RoboDK station: wcs_plc_20240513_133800.rdk

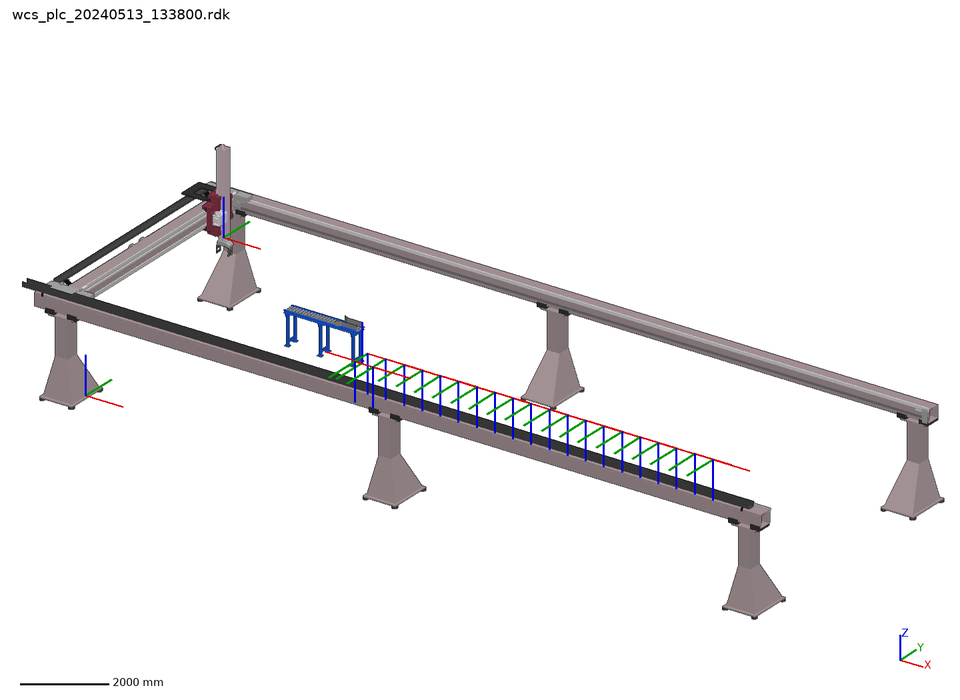
[picture v0: the station drawn from its stored meshes, robots at their saved joint values, targets as dots, program paths as lines]
Station wcs_plc_20240513_133800 (saved by RoboDK 5.6.8). Poses are relative to the parent item; angles as X-Y-Z fixed-axis rotations.
Station parameters (name, value as stored): TAGS, ['Milling']
  - frame conveyor Base IN at (4133.67, 4957.34, 0) mm, rotated rx 0 ry 0 rz 180 deg
    - robot conveyor IN: 1 axes
        modified DH rows (alpha deg, a mm, theta deg, d mm): 0, 0, 0, 0 linear
        base shift (0, 0, 0) mm, rotated rx 0 ry 90 rz 0 deg
        joint limits [-99999] to [9999999]; home [0]; saved at [1000]
      - tool conveyor_TCP_IN, TCP at (160, 110, 135) mm, rotated rx -180 ry 0 rz -180 deg
    - target con_pitch_IN (joint target) at (1000, 0, 880) mm; joints [1000, 0, 0] of conveyor IN
    - target con_home_IN (joint target) at (160, 110, 1015) mm, rotated rx -180 ry 0 rz -180 deg; joints [0] of conveyor IN
  - frame gantry Base at (0, 0, 0) mm
    - robot gantry: 3 axes
        modified DH rows (alpha deg, a mm, theta deg, d mm): 0, 0, 0, 0 linear; 90, 0, 90, 0 linear; 90, 0, 0, 0 linear
        base shift (0, 0, 0) mm, rotated rx 0 ry -90 rz 180 deg
        joint limits [-5, -5, -5] to [18000, 5000, 1500]; home [0, 0, 0]; saved at [0, 0, 0]
      - frame gripper Base at (0, 0, 0) mm, rotated rx -180 ry 0 rz 0 deg
        - robot gripper: 1 axes
            modified DH rows (alpha deg, a mm, theta deg, d mm): 0, 0, 0, 0 linear
            base shift (0, 0, 0) mm, rotated rx 0 ry 90 rz 0 deg
            joint limits [-200] to [0]; home [0]; saved at [-55]
        - target close_gripper (joint target) at (-121.33, 5507.34, 1743.56) mm; joints [-55] of gripper
        - target open_gripper (joint target) at (0, 0, 0) mm; joints [0, 0, 0] of gripper
      - tool gripper_TCP, TCP at (0, 0, 260) mm
    - target gantry_home (joint target) at (-66.33, 5507.34, 1483.56) mm, rotated rx 180 ry 0 rz 0 deg; joints [0, 0, 0] of gantry
    - target UP_pickup (joint target) at (3973.67, 4847.34, 1483.56) mm, rotated rx 180 ry 0 rz 0 deg; joints [4040, 660, 0] of gantry
    - target IN_pickup (joint target) at (3973.67, 4847.34, 1015) mm, rotated rx -180 ry 0 rz 0 deg; joints [4040, 660, 468.564] of gantry
    - target Target 6 (joint target) at (4133.67, 4957.34, 433.56) mm, rotated rx 180 ry 0 rz 0 deg; joints [4200, 550, 1050] of gantry
    - target Target 7 (Cartesian target) at (10933.67, 1007.34, 433.56) mm, rotated rx 180 ry 0 rz 0 deg; joints [11000, 4500, 1050] of gantry
    - folder pallet
      - frame TeachingPoints_01-01-01 at (4633.67, 4457.34, 568.56) mm, rotated rx 180 ry 0 rz 0 deg
        - target Point_01-01-01 (Cartesian target) at (0, 0, 0) mm; joints [4700, 1050, 915] of gantry
      - frame TeachingPoints_02-01-01 at (5133.67, 4457.34, 568.56) mm, rotated rx 180 ry 0 rz 0 deg
        - target Point_02-01-01 (Cartesian target) at (0, 0, 0) mm; joints [5200, 1050, 915] of gantry
      - frame TeachingPoints_03-01-01 at (5633.67, 4457.34, 568.56) mm, rotated rx 180 ry 0 rz 0 deg
        - target Point_03-01-01 (Cartesian target) at (0, 0, 0) mm; joints [5700, 1050, 915] of gantry
      - frame TeachingPoints_04-01-01 at (6133.67, 4457.34, 568.56) mm, rotated rx 180 ry 0 rz 0 deg
        - target Point_04-01-01 (Cartesian target) at (0, 0, 0) mm; joints [6200, 1050, 915] of gantry
      - frame TeachingPoints_05-01-01 at (6633.67, 4457.34, 568.56) mm, rotated rx 180 ry 0 rz 0 deg
        - target Point_05-01-01 (Cartesian target) at (0, 0, 0) mm; joints [6700, 1050, 915] of gantry
      - frame TeachingPoints_06-01-01 at (7133.67, 4457.34, 568.56) mm, rotated rx 180 ry 0 rz 0 deg
        - target Point_06-01-01 (Cartesian target) at (0, 0, 0) mm; joints [7200, 1050, 915] of gantry
      - frame TeachingPoints_07-01-01 at (7633.67, 4457.34, 568.56) mm, rotated rx 180 ry 0 rz 0 deg
        - target Point_07-01-01 (Cartesian target) at (0, 0, 0) mm; joints [7700, 1050, 915] of gantry
      - frame TeachingPoints_08-01-01 at (8133.67, 4457.34, 568.56) mm, rotated rx 180 ry 0 rz 0 deg
        - target Point_08-01-01 (Cartesian target) at (0, 0, 0) mm; joints [8200, 1050, 915] of gantry
      - frame TeachingPoints_09-01-01 at (8633.67, 4457.34, 568.56) mm, rotated rx 180 ry 0 rz 0 deg
        - target Point_09-01-01 (Cartesian target) at (0, 0, 0) mm; joints [8700, 1050, 915] of gantry
      - frame TeachingPoints_10-01-01 at (9133.67, 4457.34, 568.56) mm, rotated rx 180 ry 0 rz 0 deg
        - target Point_10-01-01 (Cartesian target) at (0, 0, 0) mm; joints [9200, 1050, 915] of gantry
      - frame TeachingPoints_11-01-01 at (9633.67, 4457.34, 568.56) mm, rotated rx 180 ry 0 rz 0 deg
        - target Point_11-01-01 (Cartesian target) at (0, 0, 0) mm; joints [9700, 1050, 915] of gantry
      - frame TeachingPoints_12-01-01 at (10133.67, 4457.34, 568.56) mm, rotated rx 180 ry 0 rz 0 deg
        - target Point_12-01-01 (Cartesian target) at (0, 0, 0) mm; joints [10200, 1050, 915] of gantry
      - frame TeachingPoints_13-01-01 at (10633.67, 4457.34, 568.56) mm, rotated rx 180 ry 0 rz 0 deg
        - target Point_13-01-01 (Cartesian target) at (0, 0, 0) mm; joints [10700, 1050, 915] of gantry
      - frame TeachingPoints_14-01-01 at (11133.67, 4457.34, 568.56) mm, rotated rx 180 ry 0 rz 0 deg
        - target Point_14-01-01 (Cartesian target) at (0, 0, 0) mm; joints [11200, 1050, 915] of gantry
      - frame TeachingPoints_15-01-01 at (11633.67, 4457.34, 568.56) mm, rotated rx 180 ry 0 rz 0 deg
        - target Point_15-01-01 (Cartesian target) at (0, 0, 0) mm; joints [11700, 1050, 915] of gantry
      - frame TeachingPoints_16-01-01 at (12133.67, 4457.34, 568.56) mm, rotated rx 180 ry 0 rz 0 deg
        - target Point_16-01-01 (Cartesian target) at (0, 0, 0) mm; joints [12200, 1050, 915] of gantry
      - frame TeachingPoints_17-01-01 at (12633.67, 4457.34, 568.56) mm, rotated rx 180 ry 0 rz 0 deg
        - target Point_17-01-01 (Cartesian target) at (0, 0, 0) mm; joints [12700, 1050, 915] of gantry
      - frame TeachingPoints_18-01-01 at (13133.67, 4457.34, 568.56) mm, rotated rx 180 ry 0 rz 0 deg
        - target Point_18-01-01 (Cartesian target) at (0, 0, 0) mm; joints [13200, 1050, 915] of gantry
      - frame TeachingPoints_19-01-01 at (13633.67, 4457.34, 568.56) mm, rotated rx 180 ry 0 rz 0 deg
        - target Point_19-01-01 (Cartesian target) at (0, 0, 0) mm; joints [13700, 1050, 915] of gantry
      - frame TeachingPoints_20-01-01 at (14133.67, 4457.34, 568.56) mm, rotated rx 180 ry 0 rz 0 deg
        - target Point_20-01-01 (Cartesian target) at (0, 0, 0) mm; joints [14200, 1050, 915] of gantry
      - frame TeachingPoints_01-02-01 at (4633.67, 3957.34, 568.56) mm, rotated rx 180 ry 0 rz 0 deg
        - target Point_01-02-01 (Cartesian target) at (0, 0, 0) mm; joints [4700, 1550, 915] of gantry
      - frame TeachingPoints_02-02-01 at (5133.67, 3957.34, 568.56) mm, rotated rx 180 ry 0 rz 0 deg
        - target Point_02-02-01 (Cartesian target) at (0, 0, 0) mm; joints [5200, 1550, 915] of gantry
      - frame TeachingPoints_03-02-01 at (5633.67, 3957.34, 568.56) mm, rotated rx 180 ry 0 rz 0 deg
        - target Point_03-02-01 (Cartesian target) at (0, 0, 0) mm; joints [5700, 1550, 915] of gantry
      - frame TeachingPoints_04-02-01 at (6133.67, 3957.34, 568.56) mm, rotated rx 180 ry 0 rz 0 deg
        - target Point_04-02-01 (Cartesian target) at (0, 0, 0) mm; joints [6200, 1550, 915] of gantry
      - frame TeachingPoints_05-02-01 at (6633.67, 3957.34, 568.56) mm, rotated rx 180 ry 0 rz 0 deg
        - target Point_05-02-01 (Cartesian target) at (0, 0, 0) mm; joints [6700, 1550, 915] of gantry
      - frame TeachingPoints_06-02-01 at (7133.67, 3957.34, 568.56) mm, rotated rx 180 ry 0 rz 0 deg
        - target Point_06-02-01 (Cartesian target) at (0, 0, 0) mm; joints [7200, 1550, 915] of gantry
      - frame TeachingPoints_07-02-01 at (7633.67, 3957.34, 568.56) mm, rotated rx 180 ry 0 rz 0 deg
        - target Point_07-02-01 (Cartesian target) at (0, 0, 0) mm; joints [7700, 1550, 915] of gantry
      - frame TeachingPoints_08-02-01 at (8133.67, 3957.34, 568.56) mm, rotated rx 180 ry 0 rz 0 deg
        - target Point_08-02-01 (Cartesian target) at (0, 0, 0) mm; joints [8200, 1550, 915] of gantry
      - frame TeachingPoints_09-02-01 at (8633.67, 3957.34, 568.56) mm, rotated rx 180 ry 0 rz 0 deg
        - target Point_09-02-01 (Cartesian target) at (0, 0, 0) mm; joints [8700, 1550, 915] of gantry
      - frame TeachingPoints_10-02-01 at (9133.67, 3957.34, 568.56) mm, rotated rx 180 ry 0 rz 0 deg
        - target Point_10-02-01 (Cartesian target) at (0, 0, 0) mm; joints [9200, 1550, 915] of gantry
      - frame TeachingPoints_11-02-01 at (9633.67, 3957.34, 568.56) mm, rotated rx 180 ry 0 rz 0 deg
        - target Point_11-02-01 (Cartesian target) at (0, 0, 0) mm; joints [9700, 1550, 915] of gantry
      - frame TeachingPoints_12-02-01 at (10133.67, 3957.34, 568.56) mm, rotated rx 180 ry 0 rz 0 deg
        - target Point_12-02-01 (Cartesian target) at (0, 0, 0) mm; joints [10200, 1550, 915] of gantry
      - frame TeachingPoints_13-02-01 at (10633.67, 3957.34, 568.56) mm, rotated rx 180 ry 0 rz 0 deg
        - target Point_13-02-01 (Cartesian target) at (0, 0, 0) mm; joints [10700, 1550, 915] of gantry
      - frame TeachingPoints_14-02-01 at (11133.67, 3957.34, 568.56) mm, rotated rx 180 ry 0 rz 0 deg
        - target Point_14-02-01 (Cartesian target) at (0, 0, 0) mm; joints [11200, 1550, 915] of gantry
      - frame TeachingPoints_15-02-01 at (11633.67, 3957.34, 568.56) mm, rotated rx 180 ry 0 rz 0 deg
        - target Point_15-02-01 (Cartesian target) at (0, 0, 0) mm; joints [11700, 1550, 915] of gantry
      - frame TeachingPoints_16-02-01 at (12133.67, 3957.34, 568.56) mm, rotated rx 180 ry 0 rz 0 deg
        - target Point_16-02-01 (Cartesian target) at (0, 0, 0) mm; joints [12200, 1550, 915] of gantry
      - frame TeachingPoints_17-02-01 at (12633.67, 3957.34, 568.56) mm, rotated rx 180 ry 0 rz 0 deg
        - target Point_17-02-01 (Cartesian target) at (0, 0, 0) mm; joints [12700, 1550, 915] of gantry
      - frame TeachingPoints_18-02-01 at (13133.67, 3957.34, 568.56) mm, rotated rx 180 ry 0 rz 0 deg
        - target Point_18-02-01 (Cartesian target) at (0, 0, 0) mm; joints [13200, 1550, 915] of gantry
      - frame TeachingPoints_19-02-01 at (13633.67, 3957.34, 568.56) mm, rotated rx 180 ry 0 rz 0 deg
        - target Point_19-02-01 (Cartesian target) at (0, 0, 0) mm; joints [13700, 1550, 915] of gantry
      - frame TeachingPoints_20-02-01 at (14133.67, 3957.34, 568.56) mm, rotated rx 180 ry 0 rz 0 deg
        - target Point_20-02-01 (Cartesian target) at (0, 0, 0) mm; joints [14200, 1550, 915] of gantry
      - frame TeachingPoints_01-03-01 at (4633.67, 3457.34, 568.56) mm, rotated rx 180 ry 0 rz 0 deg
        - target Point_01-03-01 (Cartesian target) at (0, 0, 0) mm; joints [4700, 2050, 915] of gantry
      - frame TeachingPoints_02-03-01 at (5133.67, 3457.34, 568.56) mm, rotated rx 180 ry 0 rz 0 deg
        - target Point_02-03-01 (Cartesian target) at (0, 0, 0) mm; joints [5200, 2050, 915] of gantry
      - frame TeachingPoints_03-03-01 at (5633.67, 3457.34, 568.56) mm, rotated rx 180 ry 0 rz 0 deg
        - target Point_03-03-01 (Cartesian target) at (0, 0, 0) mm; joints [5700, 2050, 915] of gantry
      - frame TeachingPoints_04-03-01 at (6133.67, 3457.34, 568.56) mm, rotated rx 180 ry 0 rz 0 deg
        - target Point_04-03-01 (Cartesian target) at (0, 0, 0) mm; joints [6200, 2050, 915] of gantry
      - frame TeachingPoints_05-03-01 at (6633.67, 3457.34, 568.56) mm, rotated rx 180 ry 0 rz 0 deg
        - target Point_05-03-01 (Cartesian target) at (0, 0, 0) mm; joints [6700, 2050, 915] of gantry
      - frame TeachingPoints_06-03-01 at (7133.67, 3457.34, 568.56) mm, rotated rx 180 ry 0 rz 0 deg
        - target Point_06-03-01 (Cartesian target) at (0, 0, 0) mm; joints [7200, 2050, 915] of gantry
      - frame TeachingPoints_07-03-01 at (7633.67, 3457.34, 568.56) mm, rotated rx 180 ry 0 rz 0 deg
        - target Point_07-03-01 (Cartesian target) at (0, 0, 0) mm; joints [7700, 2050, 915] of gantry
      - frame TeachingPoints_08-03-01 at (8133.67, 3457.34, 568.56) mm, rotated rx 180 ry 0 rz 0 deg
        - target Point_08-03-01 (Cartesian target) at (0, 0, 0) mm; joints [8200, 2050, 915] of gantry
      - frame TeachingPoints_09-03-01 at (8633.67, 3457.34, 568.56) mm, rotated rx 180 ry 0 rz 0 deg
        - target Point_09-03-01 (Cartesian target) at (0, 0, 0) mm; joints [8700, 2050, 915] of gantry
      - frame TeachingPoints_10-03-01 at (9133.67, 3457.34, 568.56) mm, rotated rx 180 ry 0 rz 0 deg
        - target Point_10-03-01 (Cartesian target) at (0, 0, 0) mm; joints [9200, 2050, 915] of gantry
      - frame TeachingPoints_11-03-01 at (9633.67, 3457.34, 568.56) mm, rotated rx 180 ry 0 rz 0 deg
        - target Point_11-03-01 (Cartesian target) at (0, 0, 0) mm; joints [9700, 2050, 915] of gantry
      - frame TeachingPoints_12-03-01 at (10133.67, 3457.34, 568.56) mm, rotated rx 180 ry 0 rz 0 deg
        - target Point_12-03-01 (Cartesian target) at (0, 0, 0) mm; joints [10200, 2050, 915] of gantry
      - frame TeachingPoints_13-03-01 at (10633.67, 3457.34, 568.56) mm, rotated rx 180 ry 0 rz 0 deg
        - target Point_13-03-01 (Cartesian target) at (0, 0, 0) mm; joints [10700, 2050, 915] of gantry
      - frame TeachingPoints_14-03-01 at (11133.67, 3457.34, 568.56) mm, rotated rx 180 ry 0 rz 0 deg
        - target Point_14-03-01 (Cartesian target) at (0, 0, 0) mm; joints [11200, 2050, 915] of gantry
      - frame TeachingPoints_15-03-01 at (11633.67, 3457.34, 568.56) mm, rotated rx 180 ry 0 rz 0 deg
        - target Point_15-03-01 (Cartesian target) at (0, 0, 0) mm; joints [11700, 2050, 915] of gantry
      - frame TeachingPoints_16-03-01 at (12133.67, 3457.34, 568.56) mm, rotated rx 180 ry 0 rz 0 deg
        - target Point_16-03-01 (Cartesian target) at (0, 0, 0) mm; joints [12200, 2050, 915] of gantry
      - frame TeachingPoints_17-03-01 at (12633.67, 3457.34, 568.56) mm, rotated rx 180 ry 0 rz 0 deg
        - target Point_17-03-01 (Cartesian target) at (0, 0, 0) mm; joints [12700, 2050, 915] of gantry
      - frame TeachingPoints_18-03-01 at (13133.67, 3457.34, 568.56) mm, rotated rx 180 ry 0 rz 0 deg
        - target Point_18-03-01 (Cartesian target) at (0, 0, 0) mm; joints [13200, 2050, 915] of gantry
      - frame TeachingPoints_19-03-01 at (13633.67, 3457.34, 568.56) mm, rotated rx 180 ry 0 rz 0 deg
        - target Point_19-03-01 (Cartesian target) at (0, 0, 0) mm; joints [13700, 2050, 915] of gantry
      - frame TeachingPoints_20-03-01 at (14133.67, 3457.34, 568.56) mm, rotated rx 180 ry 0 rz 0 deg
        - target Point_20-03-01 (Cartesian target) at (0, 0, 0) mm; joints [14200, 2050, 915] of gantry
      - frame TeachingPoints_01-04-01 at (4633.67, 2957.34, 568.56) mm, rotated rx 180 ry 0 rz 0 deg
        - target Point_01-04-01 (Cartesian target) at (0, 0, 0) mm; joints [4700, 2550, 915] of gantry
      - frame TeachingPoints_02-04-01 at (5133.67, 2957.34, 568.56) mm, rotated rx 180 ry 0 rz 0 deg
        - target Point_02-04-01 (Cartesian target) at (0, 0, 0) mm; joints [5200, 2550, 915] of gantry
      - frame TeachingPoints_03-04-01 at (5633.67, 2957.34, 568.56) mm, rotated rx 180 ry 0 rz 0 deg
        - target Point_03-04-01 (Cartesian target) at (0, 0, 0) mm; joints [5700, 2550, 915] of gantry
      - frame TeachingPoints_04-04-01 at (6133.67, 2957.34, 568.56) mm, rotated rx 180 ry 0 rz 0 deg
        - target Point_04-04-01 (Cartesian target) at (0, 0, 0) mm; joints [6200, 2550, 915] of gantry
      - frame TeachingPoints_05-04-01 at (6633.67, 2957.34, 568.56) mm, rotated rx 180 ry 0 rz 0 deg
        - target Point_05-04-01 (Cartesian target) at (0, 0, 0) mm; joints [6700, 2550, 915] of gantry
      - frame TeachingPoints_06-04-01 at (7133.67, 2957.34, 568.56) mm, rotated rx 180 ry 0 rz 0 deg
        - target Point_06-04-01 (Cartesian target) at (0, 0, 0) mm; joints [7200, 2550, 915] of gantry
      - frame TeachingPoints_07-04-01 at (7633.67, 2957.34, 568.56) mm, rotated rx 180 ry 0 rz 0 deg
        - target Point_07-04-01 (Cartesian target) at (0, 0, 0) mm; joints [7700, 2550, 915] of gantry
      - frame TeachingPoints_08-04-01 at (8133.67, 2957.34, 568.56) mm, rotated rx 180 ry 0 rz 0 deg
        - target Point_08-04-01 (Cartesian target) at (0, 0, 0) mm; joints [8200, 2550, 915] of gantry
      - frame TeachingPoints_09-04-01 at (8633.67, 2957.34, 568.56) mm, rotated rx 180 ry 0 rz 0 deg
        - target Point_09-04-01 (Cartesian target) at (0, 0, 0) mm; joints [8700, 2550, 915] of gantry
      - frame TeachingPoints_10-04-01 at (9133.67, 2957.34, 568.56) mm, rotated rx 180 ry 0 rz 0 deg
        - target Point_10-04-01 (Cartesian target) at (0, 0, 0) mm; joints [9200, 2550, 915] of gantry
      - frame TeachingPoints_11-04-01 at (9633.67, 2957.34, 568.56) mm, rotated rx 180 ry 0 rz 0 deg
        - target Point_11-04-01 (Cartesian target) at (0, 0, 0) mm; joints [9700, 2550, 915] of gantry
      - frame TeachingPoints_12-04-01 at (10133.67, 2957.34, 568.56) mm, rotated rx 180 ry 0 rz 0 deg
        - target Point_12-04-01 (Cartesian target) at (0, 0, 0) mm; joints [10200, 2550, 915] of gantry
      - frame TeachingPoints_13-04-01 at (10633.67, 2957.34, 568.56) mm, rotated rx 180 ry 0 rz 0 deg
        - target Point_13-04-01 (Cartesian target) at (0, 0, 0) mm; joints [10700, 2550, 915] of gantry
      - frame TeachingPoints_14-04-01 at (11133.67, 2957.34, 568.56) mm, rotated rx 180 ry 0 rz 0 deg
        - target Point_14-04-01 (Cartesian target) at (0, 0, 0) mm; joints [11200, 2550, 915] of gantry
      - frame TeachingPoints_15-04-01 at (11633.67, 2957.34, 568.56) mm, rotated rx 180 ry 0 rz 0 deg
        - target Point_15-04-01 (Cartesian target) at (0, 0, 0) mm; joints [11700, 2550, 915] of gantry
      - frame TeachingPoints_16-04-01 at (12133.67, 2957.34, 568.56) mm, rotated rx 180 ry 0 rz 0 deg
        - target Point_16-04-01 (Cartesian target) at (0, 0, 0) mm; joints [12200, 2550, 915] of gantry
      - frame TeachingPoints_17-04-01 at (12633.67, 2957.34, 568.56) mm, rotated rx 180 ry 0 rz 0 deg
        - target Point_17-04-01 (Cartesian target) at (0, 0, 0) mm; joints [12700, 2550, 915] of gantry
      - frame TeachingPoints_18-04-01 at (13133.67, 2957.34, 568.56) mm, rotated rx 180 ry 0 rz 0 deg
        - target Point_18-04-01 (Cartesian target) at (0, 0, 0) mm; joints [13200, 2550, 915] of gantry
      - frame TeachingPoints_19-04-01 at (13633.67, 2957.34, 568.56) mm, rotated rx 180 ry 0 rz 0 deg
        - target Point_19-04-01 (Cartesian target) at (0, 0, 0) mm; joints [13700, 2550, 915] of gantry
      - frame TeachingPoints_20-04-01 at (14133.67, 2957.34, 568.56) mm, rotated rx 180 ry 0 rz 0 deg
        - target Point_20-04-01 (Cartesian target) at (0, 0, 0) mm; joints [14200, 2550, 915] of gantry
      - frame TeachingPoints_01-05-01 at (4633.67, 2457.34, 568.56) mm, rotated rx 180 ry 0 rz 0 deg
        - target Point_01-05-01 (Cartesian target) at (0, 0, 0) mm; joints [4700, 3050, 915] of gantry
      - frame TeachingPoints_02-05-01 at (5133.67, 2457.34, 568.56) mm, rotated rx 180 ry 0 rz 0 deg
        - target Point_02-05-01 (Cartesian target) at (0, 0, 0) mm; joints [5200, 3050, 915] of gantry
      - frame TeachingPoints_03-05-01 at (5633.67, 2457.34, 568.56) mm, rotated rx 180 ry 0 rz 0 deg
        - target Point_03-05-01 (Cartesian target) at (0, 0, 0) mm; joints [5700, 3050, 915] of gantry
      - frame TeachingPoints_04-05-01 at (6133.67, 2457.34, 568.56) mm, rotated rx 180 ry 0 rz 0 deg
        - target Point_04-05-01 (Cartesian target) at (0, 0, 0) mm; joints [6200, 3050, 915] of gantry
      - frame TeachingPoints_05-05-01 at (6633.67, 2457.34, 568.56) mm, rotated rx 180 ry 0 rz 0 deg
        - target Point_05-05-01 (Cartesian target) at (0, 0, 0) mm; joints [6700, 3050, 915] of gantry
      - frame TeachingPoints_06-05-01 at (7133.67, 2457.34, 568.56) mm, rotated rx 180 ry 0 rz 0 deg
        - target Point_06-05-01 (Cartesian target) at (0, 0, 0) mm; joints [7200, 3050, 915] of gantry
      - frame TeachingPoints_07-05-01 at (7633.67, 2457.34, 568.56) mm, rotated rx 180 ry 0 rz 0 deg
        - target Point_07-05-01 (Cartesian target) at (0, 0, 0) mm; joints [7700, 3050, 915] of gantry
      - frame TeachingPoints_08-05-01 at (8133.67, 2457.34, 568.56) mm, rotated rx 180 ry 0 rz 0 deg
        - target Point_08-05-01 (Cartesian target) at (0, 0, 0) mm; joints [8200, 3050, 915] of gantry
      - frame TeachingPoints_09-05-01 at (8633.67, 2457.34, 568.56) mm, rotated rx 180 ry 0 rz 0 deg
        - target Point_09-05-01 (Cartesian target) at (0, 0, 0) mm; joints [8700, 3050, 915] of gantry
      - frame TeachingPoints_10-05-01 at (9133.67, 2457.34, 568.56) mm, rotated rx 180 ry 0 rz 0 deg
        - target Point_10-05-01 (Cartesian target) at (0, 0, 0) mm; joints [9200, 3050, 915] of gantry
      - frame TeachingPoints_11-05-01 at (9633.67, 2457.34, 568.56) mm, rotated rx 180 ry 0 rz 0 deg
        - target Point_11-05-01 (Cartesian target) at (0, 0, 0) mm; joints [9700, 3050, 915] of gantry
      - frame TeachingPoints_12-05-01 at (10133.67, 2457.34, 568.56) mm, rotated rx 180 ry 0 rz 0 deg
        - target Point_12-05-01 (Cartesian target) at (0, 0, 0) mm; joints [10200, 3050, 915] of gantry
      - frame TeachingPoints_13-05-01 at (10633.67, 2457.34, 568.56) mm, rotated rx 180 ry 0 rz 0 deg
        - target Point_13-05-01 (Cartesian target) at (0, 0, 0) mm; joints [10700, 3050, 915] of gantry
      - frame TeachingPoints_14-05-01 at (11133.67, 2457.34, 568.56) mm, rotated rx 180 ry 0 rz 0 deg
        - target Point_14-05-01 (Cartesian target) at (0, 0, 0) mm; joints [11200, 3050, 915] of gantry
      - frame TeachingPoints_15-05-01 at (11633.67, 2457.34, 568.56) mm, rotated rx 180 ry 0 rz 0 deg
        - target Point_15-05-01 (Cartesian target) at (0, 0, 0) mm; joints [11700, 3050, 915] of gantry
      - frame TeachingPoints_16-05-01 at (12133.67, 2457.34, 568.56) mm, rotated rx 180 ry 0 rz 0 deg
        - target Point_16-05-01 (Cartesian target) at (0, 0, 0) mm; joints [12200, 3050, 915] of gantry
      - frame TeachingPoints_17-05-01 at (12633.67, 2457.34, 568.56) mm, rotated rx 180 ry 0 rz 0 deg
        - target Point_17-05-01 (Cartesian target) at (0, 0, 0) mm; joints [12700, 3050, 915] of gantry
      - frame TeachingPoints_18-05-01 at (13133.67, 2457.34, 568.56) mm, rotated rx 180 ry 0 rz 0 deg
        - target Point_18-05-01 (Cartesian target) at (0, 0, 0) mm; joints [13200, 3050, 915] of gantry
      - frame TeachingPoints_19-05-01 at (13633.67, 2457.34, 568.56) mm, rotated rx 180 ry 0 rz 0 deg
        - target Point_19-05-01 (Cartesian target) at (0, 0, 0) mm; joints [13700, 3050, 915] of gantry
      - frame TeachingPoints_20-05-01 at (14133.67, 2457.34, 568.56) mm, rotated rx 180 ry 0 rz 0 deg
        - target Point_20-05-01 (Cartesian target) at (0, 0, 0) mm; joints [14200, 3050, 915] of gantry
      - frame TeachingPoints_01-06-01 at (4633.67, 1957.34, 568.56) mm, rotated rx 180 ry 0 rz 0 deg
        - target Point_01-06-01 (Cartesian target) at (0, 0, 0) mm; joints [4700, 3550, 915] of gantry
      - frame TeachingPoints_02-06-01 at (5133.67, 1957.34, 568.56) mm, rotated rx 180 ry 0 rz 0 deg
        - target Point_02-06-01 (Cartesian target) at (0, 0, 0) mm; joints [5200, 3550, 915] of gantry
      - frame TeachingPoints_03-06-01 at (5633.67, 1957.34, 568.56) mm, rotated rx 180 ry 0 rz 0 deg
        - target Point_03-06-01 (Cartesian target) at (0, 0, 0) mm; joints [5700, 3550, 915] of gantry
      - frame TeachingPoints_04-06-01 at (6133.67, 1957.34, 568.56) mm, rotated rx 180 ry 0 rz 0 deg
        - target Point_04-06-01 (Cartesian target) at (0, 0, 0) mm; joints [6200, 3550, 915] of gantry
      - frame TeachingPoints_05-06-01 at (6633.67, 1957.34, 568.56) mm, rotated rx 180 ry 0 rz 0 deg
        - target Point_05-06-01 (Cartesian target) at (0, 0, 0) mm; joints [6700, 3550, 915] of gantry
      - frame TeachingPoints_06-06-01 at (7133.67, 1957.34, 568.56) mm, rotated rx 180 ry 0 rz 0 deg
        - target Point_06-06-01 (Cartesian target) at (0, 0, 0) mm; joints [7200, 3550, 915] of gantry
      - frame TeachingPoints_07-06-01 at (7633.67, 1957.34, 568.56) mm, rotated rx 180 ry 0 rz 0 deg
        - target Point_07-06-01 (Cartesian target) at (0, 0, 0) mm; joints [7700, 3550, 915] of gantry
      - frame TeachingPoints_08-06-01 at (8133.67, 1957.34, 568.56) mm, rotated rx 180 ry 0 rz 0 deg
        - target Point_08-06-01 (Cartesian target) at (0, 0, 0) mm; joints [8200, 3550, 915] of gantry
      - frame TeachingPoints_09-06-01 at (8633.67, 1957.34, 568.56) mm, rotated rx 180 ry 0 rz 0 deg
        - target Point_09-06-01 (Cartesian target) at (0, 0, 0) mm; joints [8700, 3550, 915] of gantry
      - frame TeachingPoints_10-06-01 at (9133.67, 1957.34, 568.56) mm, rotated rx 180 ry 0 rz 0 deg
        - target Point_10-06-01 (Cartesian target) at (0, 0, 0) mm; joints [9200, 3550, 915] of gantry
      - frame TeachingPoints_11-06-01 at (9633.67, 1957.34, 568.56) mm, rotated rx 180 ry 0 rz 0 deg
        - target Point_11-06-01 (Cartesian target) at (0, 0, 0) mm; joints [9700, 3550, 915] of gantry
      - frame TeachingPoints_12-06-01 at (10133.67, 1957.34, 568.56) mm, rotated rx 180 ry 0 rz 0 deg
        - target Point_12-06-01 (Cartesian target) at (0, 0, 0) mm; joints [10200, 3550, 915] of gantry
      - frame TeachingPoints_13-06-01 at (10633.67, 1957.34, 568.56) mm, rotated rx 180 ry 0 rz 0 deg
        - target Point_13-06-01 (Cartesian target) at (0, 0, 0) mm; joints [10700, 3550, 915] of gantry
      - frame TeachingPoints_14-06-01 at (11133.67, 1957.34, 568.56) mm, rotated rx 180 ry 0 rz 0 deg
        - target Point_14-06-01 (Cartesian target) at (0, 0, 0) mm; joints [11200, 3550, 915] of gantry
      - frame TeachingPoints_15-06-01 at (11633.67, 1957.34, 568.56) mm, rotated rx 180 ry 0 rz 0 deg
        - target Point_15-06-01 (Cartesian target) at (0, 0, 0) mm; joints [11700, 3550, 915] of gantry
      - frame TeachingPoints_16-06-01 at (12133.67, 1957.34, 568.56) mm, rotated rx 180 ry 0 rz 0 deg
        - target Point_16-06-01 (Cartesian target) at (0, 0, 0) mm; joints [12200, 3550, 915] of gantry
      - frame TeachingPoints_17-06-01 at (12633.67, 1957.34, 568.56) mm, rotated rx 180 ry 0 rz 0 deg
        - target Point_17-06-01 (Cartesian target) at (0, 0, 0) mm; joints [12700, 3550, 915] of gantry
      - frame TeachingPoints_18-06-01 at (13133.67, 1957.34, 568.56) mm, rotated rx 180 ry 0 rz 0 deg
        - target Point_18-06-01 (Cartesian target) at (0, 0, 0) mm; joints [13200, 3550, 915] of gantry
      - frame TeachingPoints_19-06-01 at (13633.67, 1957.34, 568.56) mm, rotated rx 180 ry 0 rz 0 deg
        - target Point_19-06-01 (Cartesian target) at (0, 0, 0) mm; joints [13700, 3550, 915] of gantry
      - frame TeachingPoints_20-06-01 at (14133.67, 1957.34, 568.56) mm, rotated rx 180 ry 0 rz 0 deg
        - target Point_20-06-01 (Cartesian target) at (0, 0, 0) mm; joints [14200, 3550, 915] of gantry
      - frame TeachingPoints_01-01-02 at (4633.67, 4457.34, 703.56) mm, rotated rx 180 ry 0 rz 0 deg
        - target Point_01-01-02 (Cartesian target) at (0, 0, 0) mm; joints [4700, 1050, 780] of gantry
      - frame TeachingPoints_02-01-02 at (5133.67, 4457.34, 703.56) mm, rotated rx 180 ry 0 rz 0 deg
        - target Point_02-01-02 (Cartesian target) at (0, 0, 0) mm; joints [5200, 1050, 780] of gantry
      - frame TeachingPoints_03-01-02 at (5633.67, 4457.34, 703.56) mm, rotated rx 180 ry 0 rz 0 deg
        - target Point_03-01-02 (Cartesian target) at (0, 0, 0) mm; joints [5700, 1050, 780] of gantry
      - frame TeachingPoints_04-01-02 at (6133.67, 4457.34, 703.56) mm, rotated rx 180 ry 0 rz 0 deg
        - target Point_04-01-02 (Cartesian target) at (0, 0, 0) mm; joints [6200, 1050, 780] of gantry
      - frame TeachingPoints_05-01-02 at (6633.67, 4457.34, 703.56) mm, rotated rx 180 ry 0 rz 0 deg
        - target Point_05-01-02 (Cartesian target) at (0, 0, 0) mm; joints [6700, 1050, 780] of gantry
      - frame TeachingPoints_06-01-02 at (7133.67, 4457.34, 703.56) mm, rotated rx 180 ry 0 rz 0 deg
        - target Point_06-01-02 (Cartesian target) at (0, 0, 0) mm; joints [7200, 1050, 780] of gantry
      - frame TeachingPoints_07-01-02 at (7633.67, 4457.34, 703.56) mm, rotated rx 180 ry 0 rz 0 deg
        - target Point_07-01-02 (Cartesian target) at (0, 0, 0) mm; joints [7700, 1050, 780] of gantry
      - frame TeachingPoints_08-01-02 at (8133.67, 4457.34, 703.56) mm, rotated rx 180 ry 0 rz 0 deg
        - target Point_08-01-02 (Cartesian target) at (0, 0, 0) mm; joints [8200, 1050, 780] of gantry
      - frame TeachingPoints_09-01-02 at (8633.67, 4457.34, 703.56) mm, rotated rx 180 ry 0 rz 0 deg
        - target Point_09-01-02 (Cartesian target) at (0, 0, 0) mm; joints [8700, 1050, 780] of gantry
      - frame TeachingPoints_10-01-02 at (9133.67, 4457.34, 703.56) mm, rotated rx 180 ry 0 rz 0 deg
        - target Point_10-01-02 (Cartesian target) at (0, 0, 0) mm; joints [9200, 1050, 780] of gantry
      - frame TeachingPoints_11-01-02 at (9633.67, 4457.34, 703.56) mm, rotated rx 180 ry 0 rz 0 deg
        - target Point_11-01-02 (Cartesian target) at (0, 0, 0) mm; joints [9700, 1050, 780] of gantry
      - frame TeachingPoints_12-01-02 at (10133.67, 4457.34, 703.56) mm, rotated rx 180 ry 0 rz 0 deg
        - target Point_12-01-02 (Cartesian target) at (0, 0, 0) mm; joints [10200, 1050, 780] of gantry
      - frame TeachingPoints_13-01-02 at (10633.67, 4457.34, 703.56) mm, rotated rx 180 ry 0 rz 0 deg
        - target Point_13-01-02 (Cartesian target) at (0, 0, 0) mm; joints [10700, 1050, 780] of gantry
      - frame TeachingPoints_14-01-02 at (11133.67, 4457.34, 703.56) mm, rotated rx 180 ry 0 rz 0 deg
        - target Point_14-01-02 (Cartesian target) at (0, 0, 0) mm; joints [11200, 1050, 780] of gantry
      - frame TeachingPoints_15-01-02 at (11633.67, 4457.34, 703.56) mm, rotated rx 180 ry 0 rz 0 deg
        - target Point_15-01-02 (Cartesian target) at (0, 0, 0) mm; joints [11700, 1050, 780] of gantry
      - frame TeachingPoints_16-01-02 at (12133.67, 4457.34, 703.56) mm, rotated rx 180 ry 0 rz 0 deg
        - target Point_16-01-02 (Cartesian target) at (0, 0, 0) mm; joints [12200, 1050, 780] of gantry
      - frame TeachingPoints_17-01-02 at (12633.67, 4457.34, 703.56) mm, rotated rx 180 ry 0 rz 0 deg
        - target Point_17-01-02 (Cartesian target) at (0, 0, 0) mm; joints [12700, 1050, 780] of gantry
      - frame TeachingPoints_18-01-02 at (13133.67, 4457.34, 703.56) mm, rotated rx 180 ry 0 rz 0 deg
        - target Point_18-01-02 (Cartesian target) at (0, 0, 0) mm; joints [13200, 1050, 780] of gantry
      - frame TeachingPoints_19-01-02 at (13633.67, 4457.34, 703.56) mm, rotated rx 180 ry 0 rz 0 deg
        - target Point_19-01-02 (Cartesian target) at (0, 0, 0) mm; joints [13700, 1050, 780] of gantry
      - frame TeachingPoints_20-01-02 at (14133.67, 4457.34, 703.56) mm, rotated rx 180 ry 0 rz 0 deg
        - target Point_20-01-02 (Cartesian target) at (0, 0, 0) mm; joints [14200, 1050, 780] of gantry
      - frame TeachingPoints_01-02-02 at (4633.67, 3957.34, 703.56) mm, rotated rx 180 ry 0 rz 0 deg
        - target Point_01-02-02 (Cartesian target) at (0, 0, 0) mm; joints [4700, 1550, 780] of gantry
      - frame TeachingPoints_02-02-02 at (5133.67, 3957.34, 703.56) mm, rotated rx 180 ry 0 rz 0 deg
        - target Point_02-02-02 (Cartesian target) at (0, 0, 0) mm; joints [5200, 1550, 780] of gantry
      - frame TeachingPoints_03-02-02 at (5633.67, 3957.34, 703.56) mm, rotated rx 180 ry 0 rz 0 deg
        - target Point_03-02-02 (Cartesian target) at (0, 0, 0) mm; joints [5700, 1550, 780] of gantry
      - frame TeachingPoints_04-02-02 at (6133.67, 3957.34, 703.56) mm, rotated rx 180 ry 0 rz 0 deg
        - target Point_04-02-02 (Cartesian target) at (0, 0, 0) mm; joints [6200, 1550, 780] of gantry
      - frame TeachingPoints_05-02-02 at (6633.67, 3957.34, 703.56) mm, rotated rx 180 ry 0 rz 0 deg
        - target Point_05-02-02 (Cartesian target) at (0, 0, 0) mm; joints [6700, 1550, 780] of gantry
      - frame TeachingPoints_06-02-02 at (7133.67, 3957.34, 703.56) mm, rotated rx 180 ry 0 rz 0 deg
        - target Point_06-02-02 (Cartesian target) at (0, 0, 0) mm; joints [7200, 1550, 780] of gantry
      - frame TeachingPoints_07-02-02 at (7633.67, 3957.34, 703.56) mm, rotated rx 180 ry 0 rz 0 deg
        - target Point_07-02-02 (Cartesian target) at (0, 0, 0) mm; joints [7700, 1550, 780] of gantry
      - frame TeachingPoints_08-02-02 at (8133.67, 3957.34, 703.56) mm, rotated rx 180 ry 0 rz 0 deg
        - target Point_08-02-02 (Cartesian target) at (0, 0, 0) mm; joints [8200, 1550, 780] of gantry
      - frame TeachingPoints_09-02-02 at (8633.67, 3957.34, 703.56) mm, rotated rx 180 ry 0 rz 0 deg
        - target Point_09-02-02 (Cartesian target) at (0, 0, 0) mm; joints [8700, 1550, 780] of gantry
      - frame TeachingPoints_10-02-02 at (9133.67, 3957.34, 703.56) mm, rotated rx 180 ry 0 rz 0 deg
        - target Point_10-02-02 (Cartesian target) at (0, 0, 0) mm; joints [9200, 1550, 780] of gantry
      - frame TeachingPoints_11-02-02 at (9633.67, 3957.34, 703.56) mm, rotated rx 180 ry 0 rz 0 deg
        - target Point_11-02-02 (Cartesian target) at (0, 0, 0) mm; joints [9700, 1550, 780] of gantry
      - frame TeachingPoints_12-02-02 at (10133.67, 3957.34, 703.56) mm, rotated rx 180 ry 0 rz 0 deg
        - target Point_12-02-02 (Cartesian target) at (0, 0, 0) mm; joints [10200, 1550, 780] of gantry
      - frame TeachingPoints_13-02-02 at (10633.67, 3957.34, 703.56) mm, rotated rx 180 ry 0 rz 0 deg
        - target Point_13-02-02 (Cartesian target) at (0, 0, 0) mm; joints [10700, 1550, 780] of gantry
      - frame TeachingPoints_14-02-02 at (11133.67, 3957.34, 703.56) mm, rotated rx 180 ry 0 rz 0 deg
        - target Point_14-02-02 (Cartesian target) at (0, 0, 0) mm; joints [11200, 1550, 780] of gantry
      - frame TeachingPoints_15-02-02 at (11633.67, 3957.34, 703.56) mm, rotated rx 180 ry 0 rz 0 deg
        - target Point_15-02-02 (Cartesian target) at (0, 0, 0) mm; joints [11700, 1550, 780] of gantry
      - frame TeachingPoints_16-02-02 at (12133.67, 3957.34, 703.56) mm, rotated rx 180 ry 0 rz 0 deg
        - target Point_16-02-02 (Cartesian target) at (0, 0, 0) mm; joints [12200, 1550, 780] of gantry
      - frame TeachingPoints_17-02-02 at (12633.67, 3957.34, 703.56) mm, rotated rx 180 ry 0 rz 0 deg
        - target Point_17-02-02 (Cartesian target) at (0, 0, 0) mm; joints [12700, 1550, 780] of gantry
      - frame TeachingPoints_18-02-02 at (13133.67, 3957.34, 703.56) mm, rotated rx 180 ry 0 rz 0 deg
        - target Point_18-02-02 (Cartesian target) at (0, 0, 0) mm; joints [13200, 1550, 780] of gantry
      - frame TeachingPoints_19-02-02 at (13633.67, 3957.34, 703.56) mm, rotated rx 180 ry 0 rz 0 deg
        - target Point_19-02-02 (Cartesian target) at (0, 0, 0) mm; joints [13700, 1550, 780] of gantry
      - frame TeachingPoints_20-02-02 at (14133.67, 3957.34, 703.56) mm, rotated rx 180 ry 0 rz 0 deg
        - target Point_20-02-02 (Cartesian target) at (0, 0, 0) mm; joints [14200, 1550, 780] of gantry
      - frame TeachingPoints_01-03-02 at (4633.67, 3457.34, 703.56) mm, rotated rx 180 ry 0 rz 0 deg
        - target Point_01-03-02 (Cartesian target) at (0, 0, 0) mm; joints [4700, 2050, 780] of gantry
      - frame TeachingPoints_02-03-02 at (5133.67, 3457.34, 703.56) mm, rotated rx 180 ry 0 rz 0 deg
        - target Point_02-03-02 (Cartesian target) at (0, 0, 0) mm; joints [5200, 2050, 780] of gantry
      - frame TeachingPoints_03-03-02 at (5633.67, 3457.34, 703.56) mm, rotated rx 180 ry 0 rz 0 deg
        - target Point_03-03-02 (Cartesian target) at (0, 0, 0) mm; joints [5700, 2050, 780] of gantry
      - frame TeachingPoints_04-03-02 at (6133.67, 3457.34, 703.56) mm, rotated rx 180 ry 0 rz 0 deg
        - target Point_04-03-02 (Cartesian target) at (0, 0, 0) mm; joints [6200, 2050, 780] of gantry
      - frame TeachingPoints_05-03-02 at (6633.67, 3457.34, 703.56) mm, rotated rx 180 ry 0 rz 0 deg
        - target Point_05-03-02 (Cartesian target) at (0, 0, 0) mm; joints [6700, 2050, 780] of gantry
      - frame TeachingPoints_06-03-02 at (7133.67, 3457.34, 703.56) mm, rotated rx 180 ry 0 rz 0 deg
        - target Point_06-03-02 (Cartesian target) at (0, 0, 0) mm; joints [7200, 2050, 780] of gantry
      - frame TeachingPoints_07-03-02 at (7633.67, 3457.34, 703.56) mm, rotated rx 180 ry 0 rz 0 deg
        - target Point_07-03-02 (Cartesian target) at (0, 0, 0) mm; joints [7700, 2050, 780] of gantry
      - frame TeachingPoints_08-03-02 at (8133.67, 3457.34, 703.56) mm, rotated rx 180 ry 0 rz 0 deg
        - target Point_08-03-02 (Cartesian target) at (0, 0, 0) mm; joints [8200, 2050, 780] of gantry
      - frame TeachingPoints_09-03-02 at (8633.67, 3457.34, 703.56) mm, rotated rx 180 ry 0 rz 0 deg
        - target Point_09-03-02 (Cartesian target) at (0, 0, 0) mm; joints [8700, 2050, 780] of gantry
      - frame TeachingPoints_10-03-02 at (9133.67, 3457.34, 703.56) mm, rotated rx 180 ry 0 rz 0 deg
        - target Point_10-03-02 (Cartesian target) at (0, 0, 0) mm; joints [9200, 2050, 780] of gantry
      - frame TeachingPoints_11-03-02 at (9633.67, 3457.34, 703.56) mm, rotated rx 180 ry 0 rz 0 deg
        - target Point_11-03-02 (Cartesian target) at (0, 0, 0) mm; joints [9700, 2050, 780] of gantry
      - frame TeachingPoints_12-03-02 at (10133.67, 3457.34, 703.56) mm, rotated rx 180 ry 0 rz 0 deg
        - target Point_12-03-02 (Cartesian target) at (0, 0, 0) mm; joints [10200, 2050, 780] of gantry
      - frame TeachingPoints_13-03-02 at (10633.67, 3457.34, 703.56) mm, rotated rx 180 ry 0 rz 0 deg
        - target Point_13-03-02 (Cartesian target) at (0, 0, 0) mm; joints [10700, 2050, 780] of gantry
      - frame TeachingPoints_14-03-02 at (11133.67, 3457.34, 703.56) mm, rotated rx 180 ry 0 rz 0 deg
        - target Point_14-03-02 (Cartesian target) at (0, 0, 0) mm; joints [11200, 2050, 780] of gantry
      - frame TeachingPoints_15-03-02 at (11633.67, 3457.34, 703.56) mm, rotated rx 180 ry 0 rz 0 deg
        - target Point_15-03-02 (Cartesian target) at (0, 0, 0) mm; joints [11700, 2050, 780] of gantry
      - frame TeachingPoints_16-03-02 at (12133.67, 3457.34, 703.56) mm, rotated rx 180 ry 0 rz 0 deg
        - target Point_16-03-02 (Cartesian target) at (0, 0, 0) mm; joints [12200, 2050, 780] of gantry
      - frame TeachingPoints_17-03-02 at (12633.67, 3457.34, 703.56) mm, rotated rx 180 ry 0 rz 0 deg
        - target Point_17-03-02 (Cartesian target) at (0, 0, 0) mm; joints [12700, 2050, 780] of gantry
      - frame TeachingPoints_18-03-02 at (13133.67, 3457.34, 703.56) mm, rotated rx 180 ry 0 rz 0 deg
        - target Point_18-03-02 (Cartesian target) at (0, 0, 0) mm; joints [13200, 2050, 780] of gantry
      - frame TeachingPoints_19-03-02 at (13633.67, 3457.34, 703.56) mm, rotated rx 180 ry 0 rz 0 deg
        - target Point_19-03-02 (Cartesian target) at (0, 0, 0) mm; joints [13700, 2050, 780] of gantry
      - frame TeachingPoints_20-03-02 at (14133.67, 3457.34, 703.56) mm, rotated rx 180 ry 0 rz 0 deg
        - target Point_20-03-02 (Cartesian target) at (0, 0, 0) mm; joints [14200, 2050, 780] of gantry
      - frame TeachingPoints_01-04-02 at (4633.67, 2957.34, 703.56) mm, rotated rx 180 ry 0 rz 0 deg
        - target Point_01-04-02 (Cartesian target) at (0, 0, 0) mm; joints [4700, 2550, 780] of gantry
      - frame TeachingPoints_02-04-02 at (5133.67, 2957.34, 703.56) mm, rotated rx 180 ry 0 rz 0 deg
        - target Point_02-04-02 (Cartesian target) at (0, 0, 0) mm; joints [5200, 2550, 780] of gantry
      - frame TeachingPoints_03-04-02 at (5633.67, 2957.34, 703.56) mm, rotated rx 180 ry 0 rz 0 deg
        - target Point_03-04-02 (Cartesian target) at (0, 0, 0) mm; joints [5700, 2550, 780] of gantry
      - frame TeachingPoints_04-04-02 at (6133.67, 2957.34, 703.56) mm, rotated rx 180 ry 0 rz 0 deg
        - target Point_04-04-02 (Cartesian target) at (0, 0, 0) mm; joints [6200, 2550, 780] of gantry
      - frame TeachingPoints_05-04-02 at (6633.67, 2957.34, 703.56) mm, rotated rx 180 ry 0 rz 0 deg
        - target Point_05-04-02 (Cartesian target) at (0, 0, 0) mm; joints [6700, 2550, 780] of gantry
      - frame TeachingPoints_06-04-02 at (7133.67, 2957.34, 703.56) mm, rotated rx 180 ry 0 rz 0 deg
        - target Point_06-04-02 (Cartesian target) at (0, 0, 0) mm; joints [7200, 2550, 780] of gantry
      - frame TeachingPoints_07-04-02 at (7633.67, 2957.34, 703.56) mm, rotated rx 180 ry 0 rz 0 deg
        - target Point_07-04-02 (Cartesian target) at (0, 0, 0) mm; joints [7700, 2550, 780] of gantry
      - frame TeachingPoints_08-04-02 at (8133.67, 2957.34, 703.56) mm, rotated rx 180 ry 0 rz 0 deg
        - target Point_08-04-02 (Cartesian target) at (0, 0, 0) mm; joints [8200, 2550, 780] of gantry
      - frame TeachingPoints_09-04-02 at (8633.67, 2957.34, 703.56) mm, rotated rx 180 ry 0 rz 0 deg
        - target Point_09-04-02 (Cartesian target) at (0, 0, 0) mm; joints [8700, 2550, 780] of gantry
      - frame TeachingPoints_10-04-02 at (9133.67, 2957.34, 703.56) mm, rotated rx 180 ry 0 rz 0 deg
        - target Point_10-04-02 (Cartesian target) at (0, 0, 0) mm; joints [9200, 2550, 780] of gantry
      - frame TeachingPoints_11-04-02 at (9633.67, 2957.34, 703.56) mm, rotated rx 180 ry 0 rz 0 deg
        - target Point_11-04-02 (Cartesian target) at (0, 0, 0) mm; joints [9700, 2550, 780] of gantry
      - frame TeachingPoints_12-04-02 at (10133.67, 2957.34, 703.56) mm, rotated rx 180 ry 0 rz 0 deg
        - target Point_12-04-02 (Cartesian target) at (0, 0, 0) mm; joints [10200, 2550, 780] of gantry
      - frame TeachingPoints_13-04-02 at (10633.67, 2957.34, 703.56) mm, rotated rx 180 ry 0 rz 0 deg
        - target Point_13-04-02 (Cartesian target) at (0, 0, 0) mm; joints [10700, 2550, 780] of gantry
      - frame TeachingPoints_14-04-02 at (11133.67, 2957.34, 703.56) mm, rotated rx 180 ry 0 rz 0 deg
        - target Point_14-04-02 (Cartesian target) at (0, 0, 0) mm; joints [11200, 2550, 780] of gantry
      - frame TeachingPoints_15-04-02 at (11633.67, 2957.34, 703.56) mm, rotated rx 180 ry 0 rz 0 deg
        - target Point_15-04-02 (Cartesian target) at (0, 0, 0) mm; joints [11700, 2550, 780] of gantry
      - frame TeachingPoints_16-04-02 at (12133.67, 2957.34, 703.56) mm, rotated rx 180 ry 0 rz 0 deg
        - target Point_16-04-02 (Cartesian target) at (0, 0, 0) mm; joints [12200, 2550, 780] of gantry
      - frame TeachingPoints_17-04-02 at (12633.67, 2957.34, 703.56) mm, rotated rx 180 ry 0 rz 0 deg
        - target Point_17-04-02 (Cartesian target) at (0, 0, 0) mm; joints [12700, 2550, 780] of gantry
      - frame TeachingPoints_18-04-02 at (13133.67, 2957.34, 703.56) mm, rotated rx 180 ry 0 rz 0 deg
        - target Point_18-04-02 (Cartesian target) at (0, 0, 0) mm; joints [13200, 2550, 780] of gantry
      - frame TeachingPoints_19-04-02 at (13633.67, 2957.34, 703.56) mm, rotated rx 180 ry 0 rz 0 deg
        - target Point_19-04-02 (Cartesian target) at (0, 0, 0) mm; joints [13700, 2550, 780] of gantry
      - frame TeachingPoints_20-04-02 at (14133.67, 2957.34, 703.56) mm, rotated rx 180 ry 0 rz 0 deg
        - target Point_20-04-02 (Cartesian target) at (0, 0, 0) mm; joints [14200, 2550, 780] of gantry
      - frame TeachingPoints_01-05-02 at (4633.67, 2457.34, 703.56) mm, rotated rx 180 ry 0 rz 0 deg
        - target Point_01-05-02 (Cartesian target) at (0, 0, 0) mm; joints [4700, 3050, 780] of gantry
      - frame TeachingPoints_02-05-02 at (5133.67, 2457.34, 703.56) mm, rotated rx 180 ry 0 rz 0 deg
        - target Point_02-05-02 (Cartesian target) at (0, 0, 0) mm; joints [5200, 3050, 780] of gantry
      - frame TeachingPoints_03-05-02 at (5633.67, 2457.34, 703.56) mm, rotated rx 180 ry 0 rz 0 deg
        - target Point_03-05-02 (Cartesian target) at (0, 0, 0) mm; joints [5700, 3050, 780] of gantry
      - frame TeachingPoints_04-05-02 at (6133.67, 2457.34, 703.56) mm, rotated rx 180 ry 0 rz 0 deg
        - target Point_04-05-02 (Cartesian target) at (0, 0, 0) mm; joints [6200, 3050, 780] of gantry
      - frame TeachingPoints_05-05-02 at (6633.67, 2457.34, 703.56) mm, rotated rx 180 ry 0 rz 0 deg
        - target Point_05-05-02 (Cartesian target) at (0, 0, 0) mm; joints [6700, 3050, 780] of gantry
      - frame TeachingPoints_06-05-02 at (7133.67, 2457.34, 703.56) mm, rotated rx 180 ry 0 rz 0 deg
        - target Point_06-05-02 (Cartesian target) at (0, 0, 0) mm; joints [7200, 3050, 780] of gantry
      - frame TeachingPoints_07-05-02 at (7633.67, 2457.34, 703.56) mm, rotated rx 180 ry 0 rz 0 deg
        - target Point_07-05-02 (Cartesian target) at (0, 0, 0) mm; joints [7700, 3050, 780] of gantry
      - frame TeachingPoints_08-05-02 at (8133.67, 2457.34, 703.56) mm, rotated rx 180 ry 0 rz 0 deg
        - target Point_08-05-02 (Cartesian target) at (0, 0, 0) mm; joints [8200, 3050, 780] of gantry
      - frame TeachingPoints_09-05-02 at (8633.67, 2457.34, 703.56) mm, rotated rx 180 ry 0 rz 0 deg
        - target Point_09-05-02 (Cartesian target) at (0, 0, 0) mm; joints [8700, 3050, 780] of gantry
      - frame TeachingPoints_10-05-02 at (9133.67, 2457.34, 703.56) mm, rotated rx 180 ry 0 rz 0 deg
        - target Point_10-05-02 (Cartesian target) at (0, 0, 0) mm; joints [9200, 3050, 780] of gantry
      - frame TeachingPoints_11-05-02 at (9633.67, 2457.34, 703.56) mm, rotated rx 180 ry 0 rz 0 deg
        - target Point_11-05-02 (Cartesian target) at (0, 0, 0) mm; joints [9700, 3050, 780] of gantry
      - frame TeachingPoints_12-05-02 at (10133.67, 2457.34, 703.56) mm, rotated rx 180 ry 0 rz 0 deg
        - target Point_12-05-02 (Cartesian target) at (0, 0, 0) mm; joints [10200, 3050, 780] of gantry
      - frame TeachingPoints_13-05-02 at (10633.67, 2457.34, 703.56) mm, rotated rx 180 ry 0 rz 0 deg
        - target Point_13-05-02 (Cartesian target) at (0, 0, 0) mm; joints [10700, 3050, 780] of gantry
      - frame TeachingPoints_14-05-02 at (11133.67, 2457.34, 703.56) mm, rotated rx 180 ry 0 rz 0 deg
        - target Point_14-05-02 (Cartesian target) at (0, 0, 0) mm; joints [11200, 3050, 780] of gantry
      - frame TeachingPoints_15-05-02 at (11633.67, 2457.34, 703.56) mm, rotated rx 180 ry 0 rz 0 deg
        - target Point_15-05-02 (Cartesian target) at (0, 0, 0) mm; joints [11700, 3050, 780] of gantry
      - frame TeachingPoints_16-05-02 at (12133.67, 2457.34, 703.56) mm, rotated rx 180 ry 0 rz 0 deg
        - target Point_16-05-02 (Cartesian target) at (0, 0, 0) mm; joints [12200, 3050, 780] of gantry
      - frame TeachingPoints_17-05-02 at (12633.67, 2457.34, 703.56) mm, rotated rx 180 ry 0 rz 0 deg
        - target Point_17-05-02 (Cartesian target) at (0, 0, 0) mm; joints [12700, 3050, 780] of gantry
      - frame TeachingPoints_18-05-02 at (13133.67, 2457.34, 703.56) mm, rotated rx 180 ry 0 rz 0 deg
        - target Point_18-05-02 (Cartesian target) at (0, 0, 0) mm; joints [13200, 3050, 780] of gantry
      - frame TeachingPoints_19-05-02 at (13633.67, 2457.34, 703.56) mm, rotated rx 180 ry 0 rz 0 deg
        - target Point_19-05-02 (Cartesian target) at (0, 0, 0) mm; joints [13700, 3050, 780] of gantry
      - frame TeachingPoints_20-05-02 at (14133.67, 2457.34, 703.56) mm, rotated rx 180 ry 0 rz 0 deg
        - target Point_20-05-02 (Cartesian target) at (0, 0, 0) mm; joints [14200, 3050, 780] of gantry
      - frame TeachingPoints_01-06-02 at (4633.67, 1957.34, 703.56) mm, rotated rx 180 ry 0 rz 0 deg
        - target Point_01-06-02 (Cartesian target) at (0, 0, 0) mm; joints [4700, 3550, 780] of gantry
      - frame TeachingPoints_02-06-02 at (5133.67, 1957.34, 703.56) mm, rotated rx 180 ry 0 rz 0 deg
        - target Point_02-06-02 (Cartesian target) at (0, 0, 0) mm; joints [5200, 3550, 780] of gantry
      - frame TeachingPoints_03-06-02 at (5633.67, 1957.34, 703.56) mm, rotated rx 180 ry 0 rz 0 deg
        - target Point_03-06-02 (Cartesian target) at (0, 0, 0) mm; joints [5700, 3550, 780] of gantry
      - frame TeachingPoints_04-06-02 at (6133.67, 1957.34, 703.56) mm, rotated rx 180 ry 0 rz 0 deg
        - target Point_04-06-02 (Cartesian target) at (0, 0, 0) mm; joints [6200, 3550, 780] of gantry
      - frame TeachingPoints_05-06-02 at (6633.67, 1957.34, 703.56) mm, rotated rx 180 ry 0 rz 0 deg
        - target Point_05-06-02 (Cartesian target) at (0, 0, 0) mm; joints [6700, 3550, 780] of gantry
      - frame TeachingPoints_06-06-02 at (7133.67, 1957.34, 703.56) mm, rotated rx 180 ry 0 rz 0 deg
        - target Point_06-06-02 (Cartesian target) at (0, 0, 0) mm; joints [7200, 3550, 780] of gantry
      - frame TeachingPoints_07-06-02 at (7633.67, 1957.34, 703.56) mm, rotated rx 180 ry 0 rz 0 deg
        - target Point_07-06-02 (Cartesian target) at (0, 0, 0) mm; joints [7700, 3550, 780] of gantry
      - frame TeachingPoints_08-06-02 at (8133.67, 1957.34, 703.56) mm, rotated rx 180 ry 0 rz 0 deg
        - target Point_08-06-02 (Cartesian target) at (0, 0, 0) mm; joints [8200, 3550, 780] of gantry
      - frame TeachingPoints_09-06-02 at (8633.67, 1957.34, 703.56) mm, rotated rx 180 ry 0 rz 0 deg
        - target Point_09-06-02 (Cartesian target) at (0, 0, 0) mm; joints [8700, 3550, 780] of gantry
      - frame TeachingPoints_10-06-02 at (9133.67, 1957.34, 703.56) mm, rotated rx 180 ry 0 rz 0 deg
        - target Point_10-06-02 (Cartesian target) at (0, 0, 0) mm; joints [9200, 3550, 780] of gantry
      - frame TeachingPoints_11-06-02 at (9633.67, 1957.34, 703.56) mm, rotated rx 180 ry 0 rz 0 deg
        - target Point_11-06-02 (Cartesian target) at (0, 0, 0) mm; joints [9700, 3550, 780] of gantry
      - frame TeachingPoints_12-06-02 at (10133.67, 1957.34, 703.56) mm, rotated rx 180 ry 0 rz 0 deg
        - target Point_12-06-02 (Cartesian target) at (0, 0, 0) mm; joints [10200, 3550, 780] of gantry
      - frame TeachingPoints_13-06-02 at (10633.67, 1957.34, 703.56) mm, rotated rx 180 ry 0 rz 0 deg
        - target Point_13-06-02 (Cartesian target) at (0, 0, 0) mm; joints [10700, 3550, 780] of gantry
      - frame TeachingPoints_14-06-02 at (11133.67, 1957.34, 703.56) mm, rotated rx 180 ry 0 rz 0 deg
        - target Point_14-06-02 (Cartesian target) at (0, 0, 0) mm; joints [11200, 3550, 780] of gantry
      - frame TeachingPoints_15-06-02 at (11633.67, 1957.34, 703.56) mm, rotated rx 180 ry 0 rz 0 deg
        - target Point_15-06-02 (Cartesian target) at (0, 0, 0) mm; joints [11700, 3550, 780] of gantry
      - frame TeachingPoints_16-06-02 at (12133.67, 1957.34, 703.56) mm, rotated rx 180 ry 0 rz 0 deg
        - target Point_16-06-02 (Cartesian target) at (0, 0, 0) mm; joints [12200, 3550, 780] of gantry
      - frame TeachingPoints_17-06-02 at (12633.67, 1957.34, 703.56) mm, rotated rx 180 ry 0 rz 0 deg
        - target Point_17-06-02 (Cartesian target) at (0, 0, 0) mm; joints [12700, 3550, 780] of gantry
      - frame TeachingPoints_18-06-02 at (13133.67, 1957.34, 703.56) mm, rotated rx 180 ry 0 rz 0 deg
        - target Point_18-06-02 (Cartesian target) at (0, 0, 0) mm; joints [13200, 3550, 780] of gantry
      - frame TeachingPoints_19-06-02 at (13633.67, 1957.34, 703.56) mm, rotated rx 180 ry 0 rz 0 deg
        - target Point_19-06-02 (Cartesian target) at (0, 0, 0) mm; joints [13700, 3550, 780] of gantry
      - frame TeachingPoints_20-06-02 at (14133.67, 1957.34, 703.56) mm, rotated rx 180 ry 0 rz 0 deg
        - target Point_20-06-02 (Cartesian target) at (0, 0, 0) mm; joints [14200, 3550, 780] of gantry
      - frame TeachingPoints_01-01-03 at (4633.67, 4457.34, 838.56) mm, rotated rx 180 ry 0 rz 0 deg
        - target Point_01-01-03 (Cartesian target) at (0, 0, 0) mm; joints [4700, 1050, 645] of gantry
      - frame TeachingPoints_02-01-03 at (5133.67, 4457.34, 838.56) mm, rotated rx 180 ry 0 rz 0 deg
        - target Point_02-01-03 (Cartesian target) at (0, 0, 0) mm; joints [5200, 1050, 645] of gantry
      - frame TeachingPoints_03-01-03 at (5633.67, 4457.34, 838.56) mm, rotated rx 180 ry 0 rz 0 deg
        - target Point_03-01-03 (Cartesian target) at (0, 0, 0) mm; joints [5700, 1050, 645] of gantry
      - frame TeachingPoints_04-01-03 at (6133.67, 4457.34, 838.56) mm, rotated rx 180 ry 0 rz 0 deg
        - target Point_04-01-03 (Cartesian target) at (0, 0, 0) mm; joints [6200, 1050, 645] of gantry
      - frame TeachingPoints_05-01-03 at (6633.67, 4457.34, 838.56) mm, rotated rx 180 ry 0 rz 0 deg
        - target Point_05-01-03 (Cartesian target) at (0, 0, 0) mm; joints [6700, 1050, 645] of gantry
      - frame TeachingPoints_06-01-03 at (7133.67, 4457.34, 838.56) mm, rotated rx 180 ry 0 rz 0 deg
        - target Point_06-01-03 (Cartesian target) at (0, 0, 0) mm; joints [7200, 1050, 645] of gantry
      - frame TeachingPoints_07-01-03 at (7633.67, 4457.34, 838.56) mm, rotated rx 180 ry 0 rz 0 deg
        - target Point_07-01-03 (Cartesian target) at (0, 0, 0) mm; joints [7700, 1050, 645] of gantry
      - frame TeachingPoints_08-01-03 at (8133.67, 4457.34, 838.56) mm, rotated rx 180 ry 0 rz 0 deg
        - target Point_08-01-03 (Cartesian target) at (0, 0, 0) mm; joints [8200, 1050, 645] of gantry
      - frame TeachingPoints_09-01-03 at (8633.67, 4457.34, 838.56) mm, rotated rx 180 ry 0 rz 0 deg
        - target Point_09-01-03 (Cartesian target) at (0, 0, 0) mm; joints [8700, 1050, 645] of gantry
      - frame TeachingPoints_10-01-03 at (9133.67, 4457.34, 838.56) mm, rotated rx 180 ry 0 rz 0 deg
        - target Point_10-01-03 (Cartesian target) at (0, 0, 0) mm; joints [9200, 1050, 645] of gantry
      - frame TeachingPoints_11-01-03 at (9633.67, 4457.34, 838.56) mm, rotated rx 180 ry 0 rz 0 deg
        - target Point_11-01-03 (Cartesian target) at (0, 0, 0) mm; joints [9700, 1050, 645] of gantry
      - frame TeachingPoints_12-01-03 at (10133.67, 4457.34, 838.56) mm, rotated rx 180 ry 0 rz 0 deg
        - target Point_12-01-03 (Cartesian target) at (0, 0, 0) mm; joints [10200, 1050, 645] of gantry
      - frame TeachingPoints_13-01-03 at (10633.67, 4457.34, 838.56) mm, rotated rx 180 ry 0 rz 0 deg
        - target Point_13-01-03 (Cartesian target) at (0, 0, 0) mm; joints [10700, 1050, 645] of gantry
      - frame TeachingPoints_14-01-03 at (11133.67, 4457.34, 838.56) mm, rotated rx 180 ry 0 rz 0 deg
        - target Point_14-01-03 (Cartesian target) at (0, 0, 0) mm; joints [11200, 1050, 645] of gantry
      - frame TeachingPoints_15-01-03 at (11633.67, 4457.34, 838.56) mm, rotated rx 180 ry 0 rz 0 deg
        - target Point_15-01-03 (Cartesian target) at (0, 0, 0) mm; joints [11700, 1050, 645] of gantry
      - frame TeachingPoints_16-01-03 at (12133.67, 4457.34, 838.56) mm, rotated rx 180 ry 0 rz 0 deg
        - target Point_16-01-03 (Cartesian target) at (0, 0, 0) mm; joints [12200, 1050, 645] of gantry
      - frame TeachingPoints_17-01-03 at (12633.67, 4457.34, 838.56) mm, rotated rx 180 ry 0 rz 0 deg
        - target Point_17-01-03 (Cartesian target) at (0, 0, 0) mm; joints [12700, 1050, 645] of gantry
      - frame TeachingPoints_18-01-03 at (13133.67, 4457.34, 838.56) mm, rotated rx 180 ry 0 rz 0 deg
        - target Point_18-01-03 (Cartesian target) at (0, 0, 0) mm; joints [13200, 1050, 645] of gantry
      - frame TeachingPoints_19-01-03 at (13633.67, 4457.34, 838.56) mm, rotated rx 180 ry 0 rz 0 deg
        - target Point_19-01-03 (Cartesian target) at (0, 0, 0) mm; joints [13700, 1050, 645] of gantry
      - frame TeachingPoints_20-01-03 at (14133.67, 4457.34, 838.56) mm, rotated rx 180 ry 0 rz 0 deg
        - target Point_20-01-03 (Cartesian target) at (0, 0, 0) mm; joints [14200, 1050, 645] of gantry
      - frame TeachingPoints_01-02-03 at (4633.67, 3957.34, 838.56) mm, rotated rx 180 ry 0 rz 0 deg
        - target Point_01-02-03 (Cartesian target) at (0, 0, 0) mm; joints [4700, 1550, 645] of gantry
      - frame TeachingPoints_02-02-03 at (5133.67, 3957.34, 838.56) mm, rotated rx 180 ry 0 rz 0 deg
        - target Point_02-02-03 (Cartesian target) at (0, 0, 0) mm; joints [5200, 1550, 645] of gantry
      - frame TeachingPoints_03-02-03 at (5633.67, 3957.34, 838.56) mm, rotated rx 180 ry 0 rz 0 deg
        - target Point_03-02-03 (Cartesian target) at (0, 0, 0) mm; joints [5700, 1550, 645] of gantry
      - frame TeachingPoints_04-02-03 at (6133.67, 3957.34, 838.56) mm, rotated rx 180 ry 0 rz 0 deg
        - target Point_04-02-03 (Cartesian target) at (0, 0, 0) mm; joints [6200, 1550, 645] of gantry
      - frame TeachingPoints_05-02-03 at (6633.67, 3957.34, 838.56) mm, rotated rx 180 ry 0 rz 0 deg
        - target Point_05-02-03 (Cartesian target) at (0, 0, 0) mm; joints [6700, 1550, 645] of gantry
      - frame TeachingPoints_06-02-03 at (7133.67, 3957.34, 838.56) mm, rotated rx 180 ry 0 rz 0 deg
        - target Point_06-02-03 (Cartesian target) at (0, 0, 0) mm; joints [7200, 1550, 645] of gantry
      - frame TeachingPoints_07-02-03 at (7633.67, 3957.34, 838.56) mm, rotated rx 180 ry 0 rz 0 deg
        - target Point_07-02-03 (Cartesian target) at (0, 0, 0) mm; joints [7700, 1550, 645] of gantry
      - frame TeachingPoints_08-02-03 at (8133.67, 3957.34, 838.56) mm, rotated rx 180 ry 0 rz 0 deg
        - target Point_08-02-03 (Cartesian target) at (0, 0, 0) mm; joints [8200, 1550, 645] of gantry
      - frame TeachingPoints_09-02-03 at (8633.67, 3957.34, 838.56) mm, rotated rx 180 ry 0 rz 0 deg
        - target Point_09-02-03 (Cartesian target) at (0, 0, 0) mm; joints [8700, 1550, 645] of gantry
      - frame TeachingPoints_10-02-03 at (9133.67, 3957.34, 838.56) mm, rotated rx 180 ry 0 rz 0 deg
        - target Point_10-02-03 (Cartesian target) at (0, 0, 0) mm; joints [9200, 1550, 645] of gantry
      - frame TeachingPoints_11-02-03 at (9633.67, 3957.34, 838.56) mm, rotated rx 180 ry 0 rz 0 deg
        - target Point_11-02-03 (Cartesian target) at (0, 0, 0) mm; joints [9700, 1550, 645] of gantry
      - frame TeachingPoints_12-02-03 at (10133.67, 3957.34, 838.56) mm, rotated rx 180 ry 0 rz 0 deg
        - target Point_12-02-03 (Cartesian target) at (0, 0, 0) mm; joints [10200, 1550, 645] of gantry
      - frame TeachingPoints_13-02-03 at (10633.67, 3957.34, 838.56) mm, rotated rx 180 ry 0 rz 0 deg
        - target Point_13-02-03 (Cartesian target) at (0, 0, 0) mm; joints [10700, 1550, 645] of gantry
      - frame TeachingPoints_14-02-03 at (11133.67, 3957.34, 838.56) mm, rotated rx 180 ry 0 rz 0 deg
        - target Point_14-02-03 (Cartesian target) at (0, 0, 0) mm; joints [11200, 1550, 645] of gantry
      - frame TeachingPoints_15-02-03 at (11633.67, 3957.34, 838.56) mm, rotated rx 180 ry 0 rz 0 deg
        - target Point_15-02-03 (Cartesian target) at (0, 0, 0) mm; joints [11700, 1550, 645] of gantry
      - frame TeachingPoints_16-02-03 at (12133.67, 3957.34, 838.56) mm, rotated rx 180 ry 0 rz 0 deg
        - target Point_16-02-03 (Cartesian target) at (0, 0, 0) mm; joints [12200, 1550, 645] of gantry
      - frame TeachingPoints_17-02-03 at (12633.67, 3957.34, 838.56) mm, rotated rx 180 ry 0 rz 0 deg
        - target Point_17-02-03 (Cartesian target) at (0, 0, 0) mm; joints [12700, 1550, 645] of gantry
      - frame TeachingPoints_18-02-03 at (13133.67, 3957.34, 838.56) mm, rotated rx 180 ry 0 rz 0 deg
        - target Point_18-02-03 (Cartesian target) at (0, 0, 0) mm; joints [13200, 1550, 645] of gantry
      - frame TeachingPoints_19-02-03 at (13633.67, 3957.34, 838.56) mm, rotated rx 180 ry 0 rz 0 deg
        - target Point_19-02-03 (Cartesian target) at (0, 0, 0) mm; joints [13700, 1550, 645] of gantry
      - frame TeachingPoints_20-02-03 at (14133.67, 3957.34, 838.56) mm, rotated rx 180 ry 0 rz 0 deg
        - target Point_20-02-03 (Cartesian target) at (0, 0, 0) mm; joints [14200, 1550, 645] of gantry
      - frame TeachingPoints_01-03-03 at (4633.67, 3457.34, 838.56) mm, rotated rx 180 ry 0 rz 0 deg
        - target Point_01-03-03 (Cartesian target) at (0, 0, 0) mm; joints [4700, 2050, 645] of gantry
      - frame TeachingPoints_02-03-03 at (5133.67, 3457.34, 838.56) mm, rotated rx 180 ry 0 rz 0 deg
        - target Point_02-03-03 (Cartesian target) at (0, 0, 0) mm; joints [5200, 2050, 645] of gantry
      - frame TeachingPoints_03-03-03 at (5633.67, 3457.34, 838.56) mm, rotated rx 180 ry 0 rz 0 deg
        - target Point_03-03-03 (Cartesian target) at (0, 0, 0) mm; joints [5700, 2050, 645] of gantry
      - frame TeachingPoints_04-03-03 at (6133.67, 3457.34, 838.56) mm, rotated rx 180 ry 0 rz 0 deg
        - target Point_04-03-03 (Cartesian target) at (0, 0, 0) mm; joints [6200, 2050, 645] of gantry
      - frame TeachingPoints_05-03-03 at (6633.67, 3457.34, 838.56) mm, rotated rx 180 ry 0 rz 0 deg
        - target Point_05-03-03 (Cartesian target) at (0, 0, 0) mm; joints [6700, 2050, 645] of gantry
      - frame TeachingPoints_06-03-03 at (7133.67, 3457.34, 838.56) mm, rotated rx 180 ry 0 rz 0 deg
        - target Point_06-03-03 (Cartesian target) at (0, 0, 0) mm; joints [7200, 2050, 645] of gantry
      - frame TeachingPoints_07-03-03 at (7633.67, 3457.34, 838.56) mm, rotated rx 180 ry 0 rz 0 deg
        - target Point_07-03-03 (Cartesian target) at (0, 0, 0) mm; joints [7700, 2050, 645] of gantry
      - frame TeachingPoints_08-03-03 at (8133.67, 3457.34, 838.56) mm, rotated rx 180 ry 0 rz 0 deg
        - target Point_08-03-03 (Cartesian target) at (0, 0, 0) mm; joints [8200, 2050, 645] of gantry
      - frame TeachingPoints_09-03-03 at (8633.67, 3457.34, 838.56) mm, rotated rx 180 ry 0 rz 0 deg
        - target Point_09-03-03 (Cartesian target) at (0, 0, 0) mm; joints [8700, 2050, 645] of gantry
      - frame TeachingPoints_10-03-03 at (9133.67, 3457.34, 838.56) mm, rotated rx 180 ry 0 rz 0 deg
        - target Point_10-03-03 (Cartesian target) at (0, 0, 0) mm; joints [9200, 2050, 645] of gantry
      - frame TeachingPoints_11-03-03 at (9633.67, 3457.34, 838.56) mm, rotated rx 180 ry 0 rz 0 deg
        - target Point_11-03-03 (Cartesian target) at (0, 0, 0) mm; joints [9700, 2050, 645] of gantry
      - frame TeachingPoints_12-03-03 at (10133.67, 3457.34, 838.56) mm, rotated rx 180 ry 0 rz 0 deg
        - target Point_12-03-03 (Cartesian target) at (0, 0, 0) mm; joints [10200, 2050, 645] of gantry
      - frame TeachingPoints_13-03-03 at (10633.67, 3457.34, 838.56) mm, rotated rx 180 ry 0 rz 0 deg
        - target Point_13-03-03 (Cartesian target) at (0, 0, 0) mm; joints [10700, 2050, 645] of gantry
      - frame TeachingPoints_14-03-03 at (11133.67, 3457.34, 838.56) mm, rotated rx 180 ry 0 rz 0 deg
        - target Point_14-03-03 (Cartesian target) at (0, 0, 0) mm; joints [11200, 2050, 645] of gantry
      - frame TeachingPoints_15-03-03 at (11633.67, 3457.34, 838.56) mm, rotated rx 180 ry 0 rz 0 deg
        - target Point_15-03-03 (Cartesian target) at (0, 0, 0) mm; joints [11700, 2050, 645] of gantry
      - frame TeachingPoints_16-03-03 at (12133.67, 3457.34, 838.56) mm, rotated rx 180 ry 0 rz 0 deg
        - target Point_16-03-03 (Cartesian target) at (0, 0, 0) mm; joints [12200, 2050, 645] of gantry
      - frame TeachingPoints_17-03-03 at (12633.67, 3457.34, 838.56) mm, rotated rx 180 ry 0 rz 0 deg
        - target Point_17-03-03 (Cartesian target) at (0, 0, 0) mm; joints [12700, 2050, 645] of gantry
      - frame TeachingPoints_18-03-03 at (13133.67, 3457.34, 838.56) mm, rotated rx 180 ry 0 rz 0 deg
        - target Point_18-03-03 (Cartesian target) at (0, 0, 0) mm; joints [13200, 2050, 645] of gantry
      - frame TeachingPoints_19-03-03 at (13633.67, 3457.34, 838.56) mm, rotated rx 180 ry 0 rz 0 deg
        - target Point_19-03-03 (Cartesian target) at (0, 0, 0) mm; joints [13700, 2050, 645] of gantry
      - frame TeachingPoints_20-03-03 at (14133.67, 3457.34, 838.56) mm, rotated rx 180 ry 0 rz 0 deg
        - target Point_20-03-03 (Cartesian target) at (0, 0, 0) mm; joints [14200, 2050, 645] of gantry
      - frame TeachingPoints_01-04-03 at (4633.67, 2957.34, 838.56) mm, rotated rx 180 ry 0 rz 0 deg
        - target Point_01-04-03 (Cartesian target) at (0, 0, 0) mm; joints [4700, 2550, 645] of gantry
      - frame TeachingPoints_02-04-03 at (5133.67, 2957.34, 838.56) mm, rotated rx 180 ry 0 rz 0 deg
        - target Point_02-04-03 (Cartesian target) at (0, 0, 0) mm; joints [5200, 2550, 645] of gantry
      - frame TeachingPoints_03-04-03 at (5633.67, 2957.34, 838.56) mm, rotated rx 180 ry 0 rz 0 deg
        - target Point_03-04-03 (Cartesian target) at (0, 0, 0) mm; joints [5700, 2550, 645] of gantry
      - frame TeachingPoints_04-04-03 at (6133.67, 2957.34, 838.56) mm, rotated rx 180 ry 0 rz 0 deg
        - target Point_04-04-03 (Cartesian target) at (0, 0, 0) mm; joints [6200, 2550, 645] of gantry
      - frame TeachingPoints_05-04-03 at (6633.67, 2957.34, 838.56) mm, rotated rx 180 ry 0 rz 0 deg
        - target Point_05-04-03 (Cartesian target) at (0, 0, 0) mm; joints [6700, 2550, 645] of gantry
      - frame TeachingPoints_06-04-03 at (7133.67, 2957.34, 838.56) mm, rotated rx 180 ry 0 rz 0 deg
        - target Point_06-04-03 (Cartesian target) at (0, 0, 0) mm; joints [7200, 2550, 645] of gantry
      - frame TeachingPoints_07-04-03 at (7633.67, 2957.34, 838.56) mm, rotated rx 180 ry 0 rz 0 deg
        - target Point_07-04-03 (Cartesian target) at (0, 0, 0) mm; joints [7700, 2550, 645] of gantry
      - frame TeachingPoints_08-04-03 at (8133.67, 2957.34, 838.56) mm, rotated rx 180 ry 0 rz 0 deg
        - target Point_08-04-03 (Cartesian target) at (0, 0, 0) mm; joints [8200, 2550, 645] of gantry
      - frame TeachingPoints_09-04-03 at (8633.67, 2957.34, 838.56) mm, rotated rx 180 ry 0 rz 0 deg
        - target Point_09-04-03 (Cartesian target) at (0, 0, 0) mm; joints [8700, 2550, 645] of gantry
      - frame TeachingPoints_10-04-03 at (9133.67, 2957.34, 838.56) mm, rotated rx 180 ry 0 rz 0 deg
        - target Point_10-04-03 (Cartesian target) at (0, 0, 0) mm; joints [9200, 2550, 645] of gantry
      - frame TeachingPoints_11-04-03 at (9633.67, 2957.34, 838.56) mm, rotated rx 180 ry 0 rz 0 deg
        - target Point_11-04-03 (Cartesian target) at (0, 0, 0) mm; joints [9700, 2550, 645] of gantry
      - frame TeachingPoints_12-04-03 at (10133.67, 2957.34, 838.56) mm, rotated rx 180 ry 0 rz 0 deg
        - target Point_12-04-03 (Cartesian target) at (0, 0, 0) mm; joints [10200, 2550, 645] of gantry
      - frame TeachingPoints_13-04-03 at (10633.67, 2957.34, 838.56) mm, rotated rx 180 ry 0 rz 0 deg
        - target Point_13-04-03 (Cartesian target) at (0, 0, 0) mm; joints [10700, 2550, 645] of gantry
      - frame TeachingPoints_14-04-03 at (11133.67, 2957.34, 838.56) mm, rotated rx 180 ry 0 rz 0 deg
        - target Point_14-04-03 (Cartesian target) at (0, 0, 0) mm; joints [11200, 2550, 645] of gantry
      - frame TeachingPoints_15-04-03 at (11633.67, 2957.34, 838.56) mm, rotated rx 180 ry 0 rz 0 deg
        - target Point_15-04-03 (Cartesian target) at (0, 0, 0) mm; joints [11700, 2550, 645] of gantry
      - frame TeachingPoints_16-04-03 at (12133.67, 2957.34, 838.56) mm, rotated rx 180 ry 0 rz 0 deg
        - target Point_16-04-03 (Cartesian target) at (0, 0, 0) mm; joints [12200, 2550, 645] of gantry
      - frame TeachingPoints_17-04-03 at (12633.67, 2957.34, 838.56) mm, rotated rx 180 ry 0 rz 0 deg
        - target Point_17-04-03 (Cartesian target) at (0, 0, 0) mm; joints [12700, 2550, 645] of gantry
      - frame TeachingPoints_18-04-03 at (13133.67, 2957.34, 838.56) mm, rotated rx 180 ry 0 rz 0 deg
        - target Point_18-04-03 (Cartesian target) at (0, 0, 0) mm; joints [13200, 2550, 645] of gantry
      - frame TeachingPoints_19-04-03 at (13633.67, 2957.34, 838.56) mm, rotated rx 180 ry 0 rz 0 deg
        - target Point_19-04-03 (Cartesian target) at (0, 0, 0) mm; joints [13700, 2550, 645] of gantry
      - frame TeachingPoints_20-04-03 at (14133.67, 2957.34, 838.56) mm, rotated rx 180 ry 0 rz 0 deg
        - target Point_20-04-03 (Cartesian target) at (0, 0, 0) mm; joints [14200, 2550, 645] of gantry
      - frame TeachingPoints_01-05-03 at (4633.67, 2457.34, 838.56) mm, rotated rx 180 ry 0 rz 0 deg
        - target Point_01-05-03 (Cartesian target) at (0, 0, 0) mm; joints [4700, 3050, 645] of gantry
      - frame TeachingPoints_02-05-03 at (5133.67, 2457.34, 838.56) mm, rotated rx 180 ry 0 rz 0 deg
        - target Point_02-05-03 (Cartesian target) at (0, 0, 0) mm; joints [5200, 3050, 645] of gantry
      - frame TeachingPoints_03-05-03 at (5633.67, 2457.34, 838.56) mm, rotated rx 180 ry 0 rz 0 deg
        - target Point_03-05-03 (Cartesian target) at (0, 0, 0) mm; joints [5700, 3050, 645] of gantry
      - frame TeachingPoints_04-05-03 at (6133.67, 2457.34, 838.56) mm, rotated rx 180 ry 0 rz 0 deg
        - target Point_04-05-03 (Cartesian target) at (0, 0, 0) mm; joints [6200, 3050, 645] of gantry
      - frame TeachingPoints_05-05-03 at (6633.67, 2457.34, 838.56) mm, rotated rx 180 ry 0 rz 0 deg
        - target Point_05-05-03 (Cartesian target) at (0, 0, 0) mm; joints [6700, 3050, 645] of gantry
      - frame TeachingPoints_06-05-03 at (7133.67, 2457.34, 838.56) mm, rotated rx 180 ry 0 rz 0 deg
        - target Point_06-05-03 (Cartesian target) at (0, 0, 0) mm; joints [7200, 3050, 645] of gantry
      - frame TeachingPoints_07-05-03 at (7633.67, 2457.34, 838.56) mm, rotated rx 180 ry 0 rz 0 deg
        - target Point_07-05-03 (Cartesian target) at (0, 0, 0) mm; joints [7700, 3050, 645] of gantry
      - frame TeachingPoints_08-05-03 at (8133.67, 2457.34, 838.56) mm, rotated rx 180 ry 0 rz 0 deg
        - target Point_08-05-03 (Cartesian target) at (0, 0, 0) mm; joints [8200, 3050, 645] of gantry
      - frame TeachingPoints_09-05-03 at (8633.67, 2457.34, 838.56) mm, rotated rx 180 ry 0 rz 0 deg
        - target Point_09-05-03 (Cartesian target) at (0, 0, 0) mm; joints [8700, 3050, 645] of gantry
      - frame TeachingPoints_10-05-03 at (9133.67, 2457.34, 838.56) mm, rotated rx 180 ry 0 rz 0 deg
        - target Point_10-05-03 (Cartesian target) at (0, 0, 0) mm; joints [9200, 3050, 645] of gantry
      - frame TeachingPoints_11-05-03 at (9633.67, 2457.34, 838.56) mm, rotated rx 180 ry 0 rz 0 deg
        - target Point_11-05-03 (Cartesian target) at (0, 0, 0) mm; joints [9700, 3050, 645] of gantry
      - frame TeachingPoints_12-05-03 at (10133.67, 2457.34, 838.56) mm, rotated rx 180 ry 0 rz 0 deg
        - target Point_12-05-03 (Cartesian target) at (0, 0, 0) mm; joints [10200, 3050, 645] of gantry
      - frame TeachingPoints_13-05-03 at (10633.67, 2457.34, 838.56) mm, rotated rx 180 ry 0 rz 0 deg
        - target Point_13-05-03 (Cartesian target) at (0, 0, 0) mm; joints [10700, 3050, 645] of gantry
      - frame TeachingPoints_14-05-03 at (11133.67, 2457.34, 838.56) mm, rotated rx 180 ry 0 rz 0 deg
        - target Point_14-05-03 (Cartesian target) at (0, 0, 0) mm; joints [11200, 3050, 645] of gantry
      - frame TeachingPoints_15-05-03 at (11633.67, 2457.34, 838.56) mm, rotated rx 180 ry 0 rz 0 deg
        - target Point_15-05-03 (Cartesian target) at (0, 0, 0) mm; joints [11700, 3050, 645] of gantry
      - frame TeachingPoints_16-05-03 at (12133.67, 2457.34, 838.56) mm, rotated rx 180 ry 0 rz 0 deg
        - target Point_16-05-03 (Cartesian target) at (0, 0, 0) mm; joints [12200, 3050, 645] of gantry
      - frame TeachingPoints_17-05-03 at (12633.67, 2457.34, 838.56) mm, rotated rx 180 ry 0 rz 0 deg
        - target Point_17-05-03 (Cartesian target) at (0, 0, 0) mm; joints [12700, 3050, 645] of gantry
      - frame TeachingPoints_18-05-03 at (13133.67, 2457.34, 838.56) mm, rotated rx 180 ry 0 rz 0 deg
        - target Point_18-05-03 (Cartesian target) at (0, 0, 0) mm; joints [13200, 3050, 645] of gantry
      - frame TeachingPoints_19-05-03 at (13633.67, 2457.34, 838.56) mm, rotated rx 180 ry 0 rz 0 deg
        - target Point_19-05-03 (Cartesian target) at (0, 0, 0) mm; joints [13700, 3050, 645] of gantry
      - frame TeachingPoints_20-05-03 at (14133.67, 2457.34, 838.56) mm, rotated rx 180 ry 0 rz 0 deg
        - target Point_20-05-03 (Cartesian target) at (0, 0, 0) mm; joints [14200, 3050, 645] of gantry
      - frame TeachingPoints_01-06-03 at (4633.67, 1957.34, 838.56) mm, rotated rx 180 ry 0 rz 0 deg
        - target Point_01-06-03 (Cartesian target) at (0, 0, 0) mm; joints [4700, 3550, 645] of gantry
      - frame TeachingPoints_02-06-03 at (5133.67, 1957.34, 838.56) mm, rotated rx 180 ry 0 rz 0 deg
        - target Point_02-06-03 (Cartesian target) at (0, 0, 0) mm; joints [5200, 3550, 645] of gantry
      - frame TeachingPoints_03-06-03 at (5633.67, 1957.34, 838.56) mm, rotated rx 180 ry 0 rz 0 deg
        - target Point_03-06-03 (Cartesian target) at (0, 0, 0) mm; joints [5700, 3550, 645] of gantry
      - frame TeachingPoints_04-06-03 at (6133.67, 1957.34, 838.56) mm, rotated rx 180 ry 0 rz 0 deg
        - target Point_04-06-03 (Cartesian target) at (0, 0, 0) mm; joints [6200, 3550, 645] of gantry
      - frame TeachingPoints_05-06-03 at (6633.67, 1957.34, 838.56) mm, rotated rx 180 ry 0 rz 0 deg
        - target Point_05-06-03 (Cartesian target) at (0, 0, 0) mm; joints [6700, 3550, 645] of gantry
      - frame TeachingPoints_06-06-03 at (7133.67, 1957.34, 838.56) mm, rotated rx 180 ry 0 rz 0 deg
        - target Point_06-06-03 (Cartesian target) at (0, 0, 0) mm; joints [7200, 3550, 645] of gantry
      - frame TeachingPoints_07-06-03 at (7633.67, 1957.34, 838.56) mm, rotated rx 180 ry 0 rz 0 deg
        - target Point_07-06-03 (Cartesian target) at (0, 0, 0) mm; joints [7700, 3550, 645] of gantry
      - frame TeachingPoints_08-06-03 at (8133.67, 1957.34, 838.56) mm, rotated rx 180 ry 0 rz 0 deg
        - target Point_08-06-03 (Cartesian target) at (0, 0, 0) mm; joints [8200, 3550, 645] of gantry
      - frame TeachingPoints_09-06-03 at (8633.67, 1957.34, 838.56) mm, rotated rx 180 ry 0 rz 0 deg
        - target Point_09-06-03 (Cartesian target) at (0, 0, 0) mm; joints [8700, 3550, 645] of gantry
      - frame TeachingPoints_10-06-03 at (9133.67, 1957.34, 838.56) mm, rotated rx 180 ry 0 rz 0 deg
        - target Point_10-06-03 (Cartesian target) at (0, 0, 0) mm; joints [9200, 3550, 645] of gantry
      - frame TeachingPoints_11-06-03 at (9633.67, 1957.34, 838.56) mm, rotated rx 180 ry 0 rz 0 deg
        - target Point_11-06-03 (Cartesian target) at (0, 0, 0) mm; joints [9700, 3550, 645] of gantry
      - frame TeachingPoints_12-06-03 at (10133.67, 1957.34, 838.56) mm, rotated rx 180 ry 0 rz 0 deg
        - target Point_12-06-03 (Cartesian target) at (0, 0, 0) mm; joints [10200, 3550, 645] of gantry
      - frame TeachingPoints_13-06-03 at (10633.67, 1957.34, 838.56) mm, rotated rx 180 ry 0 rz 0 deg
        - target Point_13-06-03 (Cartesian target) at (0, 0, 0) mm; joints [10700, 3550, 645] of gantry
      - frame TeachingPoints_14-06-03 at (11133.67, 1957.34, 838.56) mm, rotated rx 180 ry 0 rz 0 deg
        - target Point_14-06-03 (Cartesian target) at (0, 0, 0) mm; joints [11200, 3550, 645] of gantry
      - frame TeachingPoints_15-06-03 at (11633.67, 1957.34, 838.56) mm, rotated rx 180 ry 0 rz 0 deg
        - target Point_15-06-03 (Cartesian target) at (0, 0, 0) mm; joints [11700, 3550, 645] of gantry
      - frame TeachingPoints_16-06-03 at (12133.67, 1957.34, 838.56) mm, rotated rx 180 ry 0 rz 0 deg
        - target Point_16-06-03 (Cartesian target) at (0, 0, 0) mm; joints [12200, 3550, 645] of gantry
      - frame TeachingPoints_17-06-03 at (12633.67, 1957.34, 838.56) mm, rotated rx 180 ry 0 rz 0 deg
        - target Point_17-06-03 (Cartesian target) at (0, 0, 0) mm; joints [12700, 3550, 645] of gantry
      - frame TeachingPoints_18-06-03 at (13133.67, 1957.34, 838.56) mm, rotated rx 180 ry 0 rz 0 deg
        - target Point_18-06-03 (Cartesian target) at (0, 0, 0) mm; joints [13200, 3550, 645] of gantry
      - frame TeachingPoints_19-06-03 at (13633.67, 1957.34, 838.56) mm, rotated rx 180 ry 0 rz 0 deg
        - target Point_19-06-03 (Cartesian target) at (0, 0, 0) mm; joints [13700, 3550, 645] of gantry
      - frame TeachingPoints_20-06-03 at (14133.67, 1957.34, 838.56) mm, rotated rx 180 ry 0 rz 0 deg
        - target Point_20-06-03 (Cartesian target) at (0, 0, 0) mm; joints [14200, 3550, 645] of gantry
      - frame TeachingPoints_01-01-04 at (4633.67, 4457.34, 973.56) mm, rotated rx 180 ry 0 rz 0 deg
        - target Point_01-01-04 (Cartesian target) at (0, 0, 0) mm; joints [4700, 1050, 510] of gantry
      - frame TeachingPoints_02-01-04 at (5133.67, 4457.34, 973.56) mm, rotated rx 180 ry 0 rz 0 deg
        - target Point_02-01-04 (Cartesian target) at (0, 0, 0) mm; joints [5200, 1050, 510] of gantry
      - frame TeachingPoints_03-01-04 at (5633.67, 4457.34, 973.56) mm, rotated rx 180 ry 0 rz 0 deg
        - target Point_03-01-04 (Cartesian target) at (0, 0, 0) mm; joints [5700, 1050, 510] of gantry
      - frame TeachingPoints_04-01-04 at (6133.67, 4457.34, 973.56) mm, rotated rx 180 ry 0 rz 0 deg
        - target Point_04-01-04 (Cartesian target) at (0, 0, 0) mm; joints [6200, 1050, 510] of gantry
      - frame TeachingPoints_05-01-04 at (6633.67, 4457.34, 973.56) mm, rotated rx 180 ry 0 rz 0 deg
        - target Point_05-01-04 (Cartesian target) at (0, 0, 0) mm; joints [6700, 1050, 510] of gantry
      - frame TeachingPoints_06-01-04 at (7133.67, 4457.34, 973.56) mm, rotated rx 180 ry 0 rz 0 deg
        - target Point_06-01-04 (Cartesian target) at (0, 0, 0) mm; joints [7200, 1050, 510] of gantry
      - frame TeachingPoints_07-01-04 at (7633.67, 4457.34, 973.56) mm, rotated rx 180 ry 0 rz 0 deg
        - target Point_07-01-04 (Cartesian target) at (0, 0, 0) mm; joints [7700, 1050, 510] of gantry
      - frame TeachingPoints_08-01-04 at (8133.67, 4457.34, 973.56) mm, rotated rx 180 ry 0 rz 0 deg
        - target Point_08-01-04 (Cartesian target) at (0, 0, 0) mm; joints [8200, 1050, 510] of gantry
      - frame TeachingPoints_09-01-04 at (8633.67, 4457.34, 973.56) mm, rotated rx 180 ry 0 rz 0 deg
        - target Point_09-01-04 (Cartesian target) at (0, 0, 0) mm; joints [8700, 1050, 510] of gantry
      - frame TeachingPoints_10-01-04 at (9133.67, 4457.34, 973.56) mm, rotated rx 180 ry 0 rz 0 deg
        - target Point_10-01-04 (Cartesian target) at (0, 0, 0) mm; joints [9200, 1050, 510] of gantry
      - frame TeachingPoints_11-01-04 at (9633.67, 4457.34, 973.56) mm, rotated rx 180 ry 0 rz 0 deg
        - target Point_11-01-04 (Cartesian target) at (0, 0, 0) mm; joints [9700, 1050, 510] of gantry
      - frame TeachingPoints_12-01-04 at (10133.67, 4457.34, 973.56) mm, rotated rx 180 ry 0 rz 0 deg
        - target Point_12-01-04 (Cartesian target) at (0, 0, 0) mm; joints [10200, 1050, 510] of gantry
      - frame TeachingPoints_13-01-04 at (10633.67, 4457.34, 973.56) mm, rotated rx 180 ry 0 rz 0 deg
        - target Point_13-01-04 (Cartesian target) at (0, 0, 0) mm; joints [10700, 1050, 510] of gantry
      - frame TeachingPoints_14-01-04 at (11133.67, 4457.34, 973.56) mm, rotated rx 180 ry 0 rz 0 deg
        - target Point_14-01-04 (Cartesian target) at (0, 0, 0) mm; joints [11200, 1050, 510] of gantry
      - frame TeachingPoints_15-01-04 at (11633.67, 4457.34, 973.56) mm, rotated rx 180 ry 0 rz 0 deg
        - target Point_15-01-04 (Cartesian target) at (0, 0, 0) mm; joints [11700, 1050, 510] of gantry
      - frame TeachingPoints_16-01-04 at (12133.67, 4457.34, 973.56) mm, rotated rx 180 ry 0 rz 0 deg
        - target Point_16-01-04 (Cartesian target) at (0, 0, 0) mm; joints [12200, 1050, 510] of gantry
      - frame TeachingPoints_17-01-04 at (12633.67, 4457.34, 973.56) mm, rotated rx 180 ry 0 rz 0 deg
        - target Point_17-01-04 (Cartesian target) at (0, 0, 0) mm; joints [12700, 1050, 510] of gantry
      - frame TeachingPoints_18-01-04 at (13133.67, 4457.34, 973.56) mm, rotated rx 180 ry 0 rz 0 deg
        - target Point_18-01-04 (Cartesian target) at (0, 0, 0) mm; joints [13200, 1050, 510] of gantry
      - frame TeachingPoints_19-01-04 at (13633.67, 4457.34, 973.56) mm, rotated rx 180 ry 0 rz 0 deg
        - target Point_19-01-04 (Cartesian target) at (0, 0, 0) mm; joints [13700, 1050, 510] of gantry
      - frame TeachingPoints_20-01-04 at (14133.67, 4457.34, 973.56) mm, rotated rx 180 ry 0 rz 0 deg
        - target Point_20-01-04 (Cartesian target) at (0, 0, 0) mm; joints [14200, 1050, 510] of gantry
      - frame TeachingPoints_01-02-04 at (4633.67, 3957.34, 973.56) mm, rotated rx 180 ry 0 rz 0 deg
        - target Point_01-02-04 (Cartesian target) at (0, 0, 0) mm; joints [4700, 1550, 510] of gantry
      - frame TeachingPoints_02-02-04 at (5133.67, 3957.34, 973.56) mm, rotated rx 180 ry 0 rz 0 deg
        - target Point_02-02-04 (Cartesian target) at (0, 0, 0) mm; joints [5200, 1550, 510] of gantry
      - frame TeachingPoints_03-02-04 at (5633.67, 3957.34, 973.56) mm, rotated rx 180 ry 0 rz 0 deg
        - target Point_03-02-04 (Cartesian target) at (0, 0, 0) mm; joints [5700, 1550, 510] of gantry
      - frame TeachingPoints_04-02-04 at (6133.67, 3957.34, 973.56) mm, rotated rx 180 ry 0 rz 0 deg
        - target Point_04-02-04 (Cartesian target) at (0, 0, 0) mm; joints [6200, 1550, 510] of gantry
      - frame TeachingPoints_05-02-04 at (6633.67, 3957.34, 973.56) mm, rotated rx 180 ry 0 rz 0 deg
        - target Point_05-02-04 (Cartesian target) at (0, 0, 0) mm; joints [6700, 1550, 510] of gantry
      - frame TeachingPoints_06-02-04 at (7133.67, 3957.34, 973.56) mm, rotated rx 180 ry 0 rz 0 deg
        - target Point_06-02-04 (Cartesian target) at (0, 0, 0) mm; joints [7200, 1550, 510] of gantry
      - frame TeachingPoints_07-02-04 at (7633.67, 3957.34, 973.56) mm, rotated rx 180 ry 0 rz 0 deg
        - target Point_07-02-04 (Cartesian target) at (0, 0, 0) mm; joints [7700, 1550, 510] of gantry
      - frame TeachingPoints_08-02-04 at (8133.67, 3957.34, 973.56) mm, rotated rx 180 ry 0 rz 0 deg
        - target Point_08-02-04 (Cartesian target) at (0, 0, 0) mm; joints [8200, 1550, 510] of gantry
      - frame TeachingPoints_09-02-04 at (8633.67, 3957.34, 973.56) mm, rotated rx 180 ry 0 rz 0 deg
        - target Point_09-02-04 (Cartesian target) at (0, 0, 0) mm; joints [8700, 1550, 510] of gantry
      - frame TeachingPoints_10-02-04 at (9133.67, 3957.34, 973.56) mm, rotated rx 180 ry 0 rz 0 deg
        - target Point_10-02-04 (Cartesian target) at (0, 0, 0) mm; joints [9200, 1550, 510] of gantry
      - frame TeachingPoints_11-02-04 at (9633.67, 3957.34, 973.56) mm, rotated rx 180 ry 0 rz 0 deg
        - target Point_11-02-04 (Cartesian target) at (0, 0, 0) mm; joints [9700, 1550, 510] of gantry
      - frame TeachingPoints_12-02-04 at (10133.67, 3957.34, 973.56) mm, rotated rx 180 ry 0 rz 0 deg
        - target Point_12-02-04 (Cartesian target) at (0, 0, 0) mm; joints [10200, 1550, 510] of gantry
      - frame TeachingPoints_13-02-04 at (10633.67, 3957.34, 973.56) mm, rotated rx 180 ry 0 rz 0 deg
        - target Point_13-02-04 (Cartesian target) at (0, 0, 0) mm; joints [10700, 1550, 510] of gantry
      - frame TeachingPoints_14-02-04 at (11133.67, 3957.34, 973.56) mm, rotated rx 180 ry 0 rz 0 deg
        - target Point_14-02-04 (Cartesian target) at (0, 0, 0) mm; joints [11200, 1550, 510] of gantry
      - frame TeachingPoints_15-02-04 at (11633.67, 3957.34, 973.56) mm, rotated rx 180 ry 0 rz 0 deg
        - target Point_15-02-04 (Cartesian target) at (0, 0, 0) mm; joints [11700, 1550, 510] of gantry
      - frame TeachingPoints_16-02-04 at (12133.67, 3957.34, 973.56) mm, rotated rx 180 ry 0 rz 0 deg
        - target Point_16-02-04 (Cartesian target) at (0, 0, 0) mm; joints [12200, 1550, 510] of gantry
      - frame TeachingPoints_17-02-04 at (12633.67, 3957.34, 973.56) mm, rotated rx 180 ry 0 rz 0 deg
        - target Point_17-02-04 (Cartesian target) at (0, 0, 0) mm; joints [12700, 1550, 510] of gantry
      - frame TeachingPoints_18-02-04 at (13133.67, 3957.34, 973.56) mm, rotated rx 180 ry 0 rz 0 deg
        - target Point_18-02-04 (Cartesian target) at (0, 0, 0) mm; joints [13200, 1550, 510] of gantry
      - frame TeachingPoints_19-02-04 at (13633.67, 3957.34, 973.56) mm, rotated rx 180 ry 0 rz 0 deg
        - target Point_19-02-04 (Cartesian target) at (0, 0, 0) mm; joints [13700, 1550, 510] of gantry
      - frame TeachingPoints_20-02-04 at (14133.67, 3957.34, 973.56) mm, rotated rx 180 ry 0 rz 0 deg
        - target Point_20-02-04 (Cartesian target) at (0, 0, 0) mm; joints [14200, 1550, 510] of gantry
      - frame TeachingPoints_01-03-04 at (4633.67, 3457.34, 973.56) mm, rotated rx 180 ry 0 rz 0 deg
        - target Point_01-03-04 (Cartesian target) at (0, 0, 0) mm; joints [4700, 2050, 510] of gantry
      - frame TeachingPoints_02-03-04 at (5133.67, 3457.34, 973.56) mm, rotated rx 180 ry 0 rz 0 deg
        - target Point_02-03-04 (Cartesian target) at (0, 0, 0) mm; joints [5200, 2050, 510] of gantry
      - frame TeachingPoints_03-03-04 at (5633.67, 3457.34, 973.56) mm, rotated rx 180 ry 0 rz 0 deg
        - target Point_03-03-04 (Cartesian target) at (0, 0, 0) mm; joints [5700, 2050, 510] of gantry
      - frame TeachingPoints_04-03-04 at (6133.67, 3457.34, 973.56) mm, rotated rx 180 ry 0 rz 0 deg
        - target Point_04-03-04 (Cartesian target) at (0, 0, 0) mm; joints [6200, 2050, 510] of gantry
      - frame TeachingPoints_05-03-04 at (6633.67, 3457.34, 973.56) mm, rotated rx 180 ry 0 rz 0 deg
        - target Point_05-03-04 (Cartesian target) at (0, 0, 0) mm; joints [6700, 2050, 510] of gantry
      - frame TeachingPoints_06-03-04 at (7133.67, 3457.34, 973.56) mm, rotated rx 180 ry 0 rz 0 deg
        - target Point_06-03-04 (Cartesian target) at (0, 0, 0) mm; joints [7200, 2050, 510] of gantry
      - frame TeachingPoints_07-03-04 at (7633.67, 3457.34, 973.56) mm, rotated rx 180 ry 0 rz 0 deg
        - target Point_07-03-04 (Cartesian target) at (0, 0, 0) mm; joints [7700, 2050, 510] of gantry
      - frame TeachingPoints_08-03-04 at (8133.67, 3457.34, 973.56) mm, rotated rx 180 ry 0 rz 0 deg
        - target Point_08-03-04 (Cartesian target) at (0, 0, 0) mm; joints [8200, 2050, 510] of gantry
      - frame TeachingPoints_09-03-04 at (8633.67, 3457.34, 973.56) mm, rotated rx 180 ry 0 rz 0 deg
        - target Point_09-03-04 (Cartesian target) at (0, 0, 0) mm; joints [8700, 2050, 510] of gantry
      - frame TeachingPoints_10-03-04 at (9133.67, 3457.34, 973.56) mm, rotated rx 180 ry 0 rz 0 deg
        - target Point_10-03-04 (Cartesian target) at (0, 0, 0) mm; joints [9200, 2050, 510] of gantry
      - frame TeachingPoints_11-03-04 at (9633.67, 3457.34, 973.56) mm, rotated rx 180 ry 0 rz 0 deg
        - target Point_11-03-04 (Cartesian target) at (0, 0, 0) mm; joints [9700, 2050, 510] of gantry
      - frame TeachingPoints_12-03-04 at (10133.67, 3457.34, 973.56) mm, rotated rx 180 ry 0 rz 0 deg
        - target Point_12-03-04 (Cartesian target) at (0, 0, 0) mm; joints [10200, 2050, 510] of gantry
      - frame TeachingPoints_13-03-04 at (10633.67, 3457.34, 973.56) mm, rotated rx 180 ry 0 rz 0 deg
        - target Point_13-03-04 (Cartesian target) at (0, 0, 0) mm; joints [10700, 2050, 510] of gantry
      - frame TeachingPoints_14-03-04 at (11133.67, 3457.34, 973.56) mm, rotated rx 180 ry 0 rz 0 deg
        - target Point_14-03-04 (Cartesian target) at (0, 0, 0) mm; joints [11200, 2050, 510] of gantry
      - frame TeachingPoints_15-03-04 at (11633.67, 3457.34, 973.56) mm, rotated rx 180 ry 0 rz 0 deg
        - target Point_15-03-04 (Cartesian target) at (0, 0, 0) mm; joints [11700, 2050, 510] of gantry
      - frame TeachingPoints_16-03-04 at (12133.67, 3457.34, 973.56) mm, rotated rx 180 ry 0 rz 0 deg
        - target Point_16-03-04 (Cartesian target) at (0, 0, 0) mm; joints [12200, 2050, 510] of gantry
      - frame TeachingPoints_17-03-04 at (12633.67, 3457.34, 973.56) mm, rotated rx 180 ry 0 rz 0 deg
        - target Point_17-03-04 (Cartesian target) at (0, 0, 0) mm; joints [12700, 2050, 510] of gantry
      - frame TeachingPoints_18-03-04 at (13133.67, 3457.34, 973.56) mm, rotated rx 180 ry 0 rz 0 deg
        - target Point_18-03-04 (Cartesian target) at (0, 0, 0) mm; joints [13200, 2050, 510] of gantry
      - frame TeachingPoints_19-03-04 at (13633.67, 3457.34, 973.56) mm, rotated rx 180 ry 0 rz 0 deg
        - target Point_19-03-04 (Cartesian target) at (0, 0, 0) mm; joints [13700, 2050, 510] of gantry
      - frame TeachingPoints_20-03-04 at (14133.67, 3457.34, 973.56) mm, rotated rx 180 ry 0 rz 0 deg
        - target Point_20-03-04 (Cartesian target) at (0, 0, 0) mm; joints [14200, 2050, 510] of gantry
      - frame TeachingPoints_01-04-04 at (4633.67, 2957.34, 973.56) mm, rotated rx 180 ry 0 rz 0 deg
        - target Point_01-04-04 (Cartesian target) at (0, 0, 0) mm; joints [4700, 2550, 510] of gantry
      - frame TeachingPoints_02-04-04 at (5133.67, 2957.34, 973.56) mm, rotated rx 180 ry 0 rz 0 deg
        - target Point_02-04-04 (Cartesian target) at (0, 0, 0) mm; joints [5200, 2550, 510] of gantry
      - frame TeachingPoints_03-04-04 at (5633.67, 2957.34, 973.56) mm, rotated rx 180 ry 0 rz 0 deg
        - target Point_03-04-04 (Cartesian target) at (0, 0, 0) mm; joints [5700, 2550, 510] of gantry
      - frame TeachingPoints_04-04-04 at (6133.67, 2957.34, 973.56) mm, rotated rx 180 ry 0 rz 0 deg
        - target Point_04-04-04 (Cartesian target) at (0, 0, 0) mm; joints [6200, 2550, 510] of gantry
      - frame TeachingPoints_05-04-04 at (6633.67, 2957.34, 973.56) mm, rotated rx 180 ry 0 rz 0 deg
        - target Point_05-04-04 (Cartesian target) at (0, 0, 0) mm; joints [6700, 2550, 510] of gantry
      - frame TeachingPoints_06-04-04 at (7133.67, 2957.34, 973.56) mm, rotated rx 180 ry 0 rz 0 deg
        - target Point_06-04-04 (Cartesian target) at (0, 0, 0) mm; joints [7200, 2550, 510] of gantry
      - frame TeachingPoints_07-04-04 at (7633.67, 2957.34, 973.56) mm, rotated rx 180 ry 0 rz 0 deg
        - target Point_07-04-04 (Cartesian target) at (0, 0, 0) mm; joints [7700, 2550, 510] of gantry
      - frame TeachingPoints_08-04-04 at (8133.67, 2957.34, 973.56) mm, rotated rx 180 ry 0 rz 0 deg
        - target Point_08-04-04 (Cartesian target) at (0, 0, 0) mm; joints [8200, 2550, 510] of gantry
      - frame TeachingPoints_09-04-04 at (8633.67, 2957.34, 973.56) mm, rotated rx 180 ry 0 rz 0 deg
        - target Point_09-04-04 (Cartesian target) at (0, 0, 0) mm; joints [8700, 2550, 510] of gantry
      - frame TeachingPoints_10-04-04 at (9133.67, 2957.34, 973.56) mm, rotated rx 180 ry 0 rz 0 deg
        - target Point_10-04-04 (Cartesian target) at (0, 0, 0) mm; joints [9200, 2550, 510] of gantry
      - frame TeachingPoints_11-04-04 at (9633.67, 2957.34, 973.56) mm, rotated rx 180 ry 0 rz 0 deg
        - target Point_11-04-04 (Cartesian target) at (0, 0, 0) mm; joints [9700, 2550, 510] of gantry
      - frame TeachingPoints_12-04-04 at (10133.67, 2957.34, 973.56) mm, rotated rx 180 ry 0 rz 0 deg
        - target Point_12-04-04 (Cartesian target) at (0, 0, 0) mm; joints [10200, 2550, 510] of gantry
      - frame TeachingPoints_13-04-04 at (10633.67, 2957.34, 973.56) mm, rotated rx 180 ry 0 rz 0 deg
        - target Point_13-04-04 (Cartesian target) at (0, 0, 0) mm; joints [10700, 2550, 510] of gantry
      - frame TeachingPoints_14-04-04 at (11133.67, 2957.34, 973.56) mm, rotated rx 180 ry 0 rz 0 deg
        - target Point_14-04-04 (Cartesian target) at (0, 0, 0) mm; joints [11200, 2550, 510] of gantry
      - frame TeachingPoints_15-04-04 at (11633.67, 2957.34, 973.56) mm, rotated rx 180 ry 0 rz 0 deg
        - target Point_15-04-04 (Cartesian target) at (0, 0, 0) mm; joints [11700, 2550, 510] of gantry
      - frame TeachingPoints_16-04-04 at (12133.67, 2957.34, 973.56) mm, rotated rx 180 ry 0 rz 0 deg
        - target Point_16-04-04 (Cartesian target) at (0, 0, 0) mm; joints [12200, 2550, 510] of gantry
      - frame TeachingPoints_17-04-04 at (12633.67, 2957.34, 973.56) mm, rotated rx 180 ry 0 rz 0 deg
        - target Point_17-04-04 (Cartesian target) at (0, 0, 0) mm; joints [12700, 2550, 510] of gantry
      - frame TeachingPoints_18-04-04 at (13133.67, 2957.34, 973.56) mm, rotated rx 180 ry 0 rz 0 deg
        - target Point_18-04-04 (Cartesian target) at (0, 0, 0) mm; joints [13200, 2550, 510] of gantry
      - frame TeachingPoints_19-04-04 at (13633.67, 2957.34, 973.56) mm, rotated rx 180 ry 0 rz 0 deg
        - target Point_19-04-04 (Cartesian target) at (0, 0, 0) mm; joints [13700, 2550, 510] of gantry
      - frame TeachingPoints_20-04-04 at (14133.67, 2957.34, 973.56) mm, rotated rx 180 ry 0 rz 0 deg
        - target Point_20-04-04 (Cartesian target) at (0, 0, 0) mm; joints [14200, 2550, 510] of gantry
      - frame TeachingPoints_01-05-04 at (4633.67, 2457.34, 973.56) mm, rotated rx 180 ry 0 rz 0 deg
        - target Point_01-05-04 (Cartesian target) at (0, 0, 0) mm; joints [4700, 3050, 510] of gantry
      - frame TeachingPoints_02-05-04 at (5133.67, 2457.34, 973.56) mm, rotated rx 180 ry 0 rz 0 deg
        - target Point_02-05-04 (Cartesian target) at (0, 0, 0) mm; joints [5200, 3050, 510] of gantry
      - frame TeachingPoints_03-05-04 at (5633.67, 2457.34, 973.56) mm, rotated rx 180 ry 0 rz 0 deg
        - target Point_03-05-04 (Cartesian target) at (0, 0, 0) mm; joints [5700, 3050, 510] of gantry
      - frame TeachingPoints_04-05-04 at (6133.67, 2457.34, 973.56) mm, rotated rx 180 ry 0 rz 0 deg
        - target Point_04-05-04 (Cartesian target) at (0, 0, 0) mm; joints [6200, 3050, 510] of gantry
      - frame TeachingPoints_05-05-04 at (6633.67, 2457.34, 973.56) mm, rotated rx 180 ry 0 rz 0 deg
        - target Point_05-05-04 (Cartesian target) at (0, 0, 0) mm; joints [6700, 3050, 510] of gantry
      - frame TeachingPoints_06-05-04 at (7133.67, 2457.34, 973.56) mm, rotated rx 180 ry 0 rz 0 deg
        - target Point_06-05-04 (Cartesian target) at (0, 0, 0) mm; joints [7200, 3050, 510] of gantry
      - frame TeachingPoints_07-05-04 at (7633.67, 2457.34, 973.56) mm, rotated rx 180 ry 0 rz 0 deg
        - target Point_07-05-04 (Cartesian target) at (0, 0, 0) mm; joints [7700, 3050, 510] of gantry
      - frame TeachingPoints_08-05-04 at (8133.67, 2457.34, 973.56) mm, rotated rx 180 ry 0 rz 0 deg
        - target Point_08-05-04 (Cartesian target) at (0, 0, 0) mm; joints [8200, 3050, 510] of gantry
      - frame TeachingPoints_09-05-04 at (8633.67, 2457.34, 973.56) mm, rotated rx 180 ry 0 rz 0 deg
        - target Point_09-05-04 (Cartesian target) at (0, 0, 0) mm; joints [8700, 3050, 510] of gantry
      - frame TeachingPoints_10-05-04 at (9133.67, 2457.34, 973.56) mm, rotated rx 180 ry 0 rz 0 deg
        - target Point_10-05-04 (Cartesian target) at (0, 0, 0) mm; joints [9200, 3050, 510] of gantry
      - frame TeachingPoints_11-05-04 at (9633.67, 2457.34, 973.56) mm, rotated rx 180 ry 0 rz 0 deg
        - target Point_11-05-04 (Cartesian target) at (0, 0, 0) mm; joints [9700, 3050, 510] of gantry
      - frame TeachingPoints_12-05-04 at (10133.67, 2457.34, 973.56) mm, rotated rx 180 ry 0 rz 0 deg
        - target Point_12-05-04 (Cartesian target) at (0, 0, 0) mm; joints [10200, 3050, 510] of gantry
      - frame TeachingPoints_13-05-04 at (10633.67, 2457.34, 973.56) mm, rotated rx 180 ry 0 rz 0 deg
        - target Point_13-05-04 (Cartesian target) at (0, 0, 0) mm; joints [10700, 3050, 510] of gantry
      - frame TeachingPoints_14-05-04 at (11133.67, 2457.34, 973.56) mm, rotated rx 180 ry 0 rz 0 deg
        - target Point_14-05-04 (Cartesian target) at (0, 0, 0) mm; joints [11200, 3050, 510] of gantry
      - frame TeachingPoints_15-05-04 at (11633.67, 2457.34, 973.56) mm, rotated rx 180 ry 0 rz 0 deg
        - target Point_15-05-04 (Cartesian target) at (0, 0, 0) mm; joints [11700, 3050, 510] of gantry
      - frame TeachingPoints_16-05-04 at (12133.67, 2457.34, 973.56) mm, rotated rx 180 ry 0 rz 0 deg
        - target Point_16-05-04 (Cartesian target) at (0, 0, 0) mm; joints [12200, 3050, 510] of gantry
      - frame TeachingPoints_17-05-04 at (12633.67, 2457.34, 973.56) mm, rotated rx 180 ry 0 rz 0 deg
        - target Point_17-05-04 (Cartesian target) at (0, 0, 0) mm; joints [12700, 3050, 510] of gantry
      - frame TeachingPoints_18-05-04 at (13133.67, 2457.34, 973.56) mm, rotated rx 180 ry 0 rz 0 deg
        - target Point_18-05-04 (Cartesian target) at (0, 0, 0) mm; joints [13200, 3050, 510] of gantry
      - frame TeachingPoints_19-05-04 at (13633.67, 2457.34, 973.56) mm, rotated rx 180 ry 0 rz 0 deg
        - target Point_19-05-04 (Cartesian target) at (0, 0, 0) mm; joints [13700, 3050, 510] of gantry
      - frame TeachingPoints_20-05-04 at (14133.67, 2457.34, 973.56) mm, rotated rx 180 ry 0 rz 0 deg
        - target Point_20-05-04 (Cartesian target) at (0, 0, 0) mm; joints [14200, 3050, 510] of gantry
      - frame TeachingPoints_01-06-04 at (4633.67, 1957.34, 973.56) mm, rotated rx 180 ry 0 rz 0 deg
        - target Point_01-06-04 (Cartesian target) at (0, 0, 0) mm; joints [4700, 3550, 510] of gantry
      - frame TeachingPoints_02-06-04 at (5133.67, 1957.34, 973.56) mm, rotated rx 180 ry 0 rz 0 deg
        - target Point_02-06-04 (Cartesian target) at (0, 0, 0) mm; joints [5200, 3550, 510] of gantry
      - frame TeachingPoints_03-06-04 at (5633.67, 1957.34, 973.56) mm, rotated rx 180 ry 0 rz 0 deg
        - target Point_03-06-04 (Cartesian target) at (0, 0, 0) mm; joints [5700, 3550, 510] of gantry
      - frame TeachingPoints_04-06-04 at (6133.67, 1957.34, 973.56) mm, rotated rx 180 ry 0 rz 0 deg
        - target Point_04-06-04 (Cartesian target) at (0, 0, 0) mm; joints [6200, 3550, 510] of gantry
      - frame TeachingPoints_05-06-04 at (6633.67, 1957.34, 973.56) mm, rotated rx 180 ry 0 rz 0 deg
        - target Point_05-06-04 (Cartesian target) at (0, 0, 0) mm; joints [6700, 3550, 510] of gantry
      - frame TeachingPoints_06-06-04 at (7133.67, 1957.34, 973.56) mm, rotated rx 180 ry 0 rz 0 deg
        - target Point_06-06-04 (Cartesian target) at (0, 0, 0) mm; joints [7200, 3550, 510] of gantry
      - frame TeachingPoints_07-06-04 at (7633.67, 1957.34, 973.56) mm, rotated rx 180 ry 0 rz 0 deg
        - target Point_07-06-04 (Cartesian target) at (0, 0, 0) mm; joints [7700, 3550, 510] of gantry
      - frame TeachingPoints_08-06-04 at (8133.67, 1957.34, 973.56) mm, rotated rx 180 ry 0 rz 0 deg
        - target Point_08-06-04 (Cartesian target) at (0, 0, 0) mm; joints [8200, 3550, 510] of gantry
      - frame TeachingPoints_09-06-04 at (8633.67, 1957.34, 973.56) mm, rotated rx 180 ry 0 rz 0 deg
        - target Point_09-06-04 (Cartesian target) at (0, 0, 0) mm; joints [8700, 3550, 510] of gantry
      - frame TeachingPoints_10-06-04 at (9133.67, 1957.34, 973.56) mm, rotated rx 180 ry 0 rz 0 deg
        - target Point_10-06-04 (Cartesian target) at (0, 0, 0) mm; joints [9200, 3550, 510] of gantry
      - frame TeachingPoints_11-06-04 at (9633.67, 1957.34, 973.56) mm, rotated rx 180 ry 0 rz 0 deg
        - target Point_11-06-04 (Cartesian target) at (0, 0, 0) mm; joints [9700, 3550, 510] of gantry
      - frame TeachingPoints_12-06-04 at (10133.67, 1957.34, 973.56) mm, rotated rx 180 ry 0 rz 0 deg
        - target Point_12-06-04 (Cartesian target) at (0, 0, 0) mm; joints [10200, 3550, 510] of gantry
      - frame TeachingPoints_13-06-04 at (10633.67, 1957.34, 973.56) mm, rotated rx 180 ry 0 rz 0 deg
        - target Point_13-06-04 (Cartesian target) at (0, 0, 0) mm; joints [10700, 3550, 510] of gantry
      - frame TeachingPoints_14-06-04 at (11133.67, 1957.34, 973.56) mm, rotated rx 180 ry 0 rz 0 deg
        - target Point_14-06-04 (Cartesian target) at (0, 0, 0) mm; joints [11200, 3550, 510] of gantry
      - frame TeachingPoints_15-06-04 at (11633.67, 1957.34, 973.56) mm, rotated rx 180 ry 0 rz 0 deg
        - target Point_15-06-04 (Cartesian target) at (0, 0, 0) mm; joints [11700, 3550, 510] of gantry
